Fanuc TP program (LS listing): op5_med_master_air_c.ls

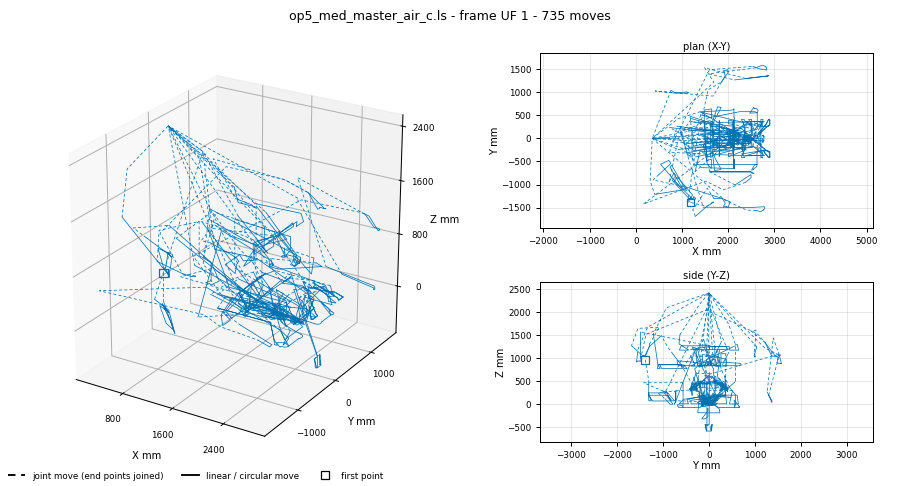
[picture p0: tool path of op5_med_master_air_c.ls in frame UF 1, 735 of 735 moves have a stored position in this frame; points joined in program order, loops and branches not executed]
/PROG  OP5_MED_MASTER_AIR_C
/ATTR
OWNER		= MNEDITOR;
COMMENT		= "Medium Main Air";
PROG_SIZE	= 94128;
CREATE		= DATE 25-08-22  TIME 11:43:26;
MODIFIED	= DATE 26-02-10  TIME 12:20:08;
FILE_NAME	= OP5_MED_;
VERSION		= 0;
LINE_COUNT	= 2444;
MEMORY_SIZE	= 94772;
PROTECT		= READ_WRITE;
TCD:  STACK_SIZE	= 0,
      TASK_PRIORITY	= 50,
      TIME_SLICE	= 0,
      BUSY_LAMP_OFF	= 0,
      ABORT_REQUEST	= 0,
      PAUSE_REQUEST	= 0;
DEFAULT_GROUP	= 1,1,*,*,*;
CONTROL_CODE	= 00000000 00000000;
/APPL
  ARC Welding Equipment : 1,*,*,*,*;

MPAS ;
MPAS_NUM_PASSES        : 0;
MPAS_LAST_PASS         : 0;
MPAS_CURRENT_PASS      : 0;
MPAS_STATUS_PASS       : 0;
/MN
   1:  !********** WAR HAMMER ********** ;
   2:  !*------- FRAME MEIDIUM --------* ;
   3:  !*------- FR500 CELL: C --------* ;
   4:  !******************************** ;
   5:   ;
   6:  CALL HOME    ;
   7:  UFRAME_NUM=1 ;
   8:   ;
   9:  !********POSITIONER MOVE******** ;
  10:J P[1] 85% CNT70    ;
  11:   ;
  12:J P[2] 50% CNT50    ;
  13:   ;
  14:L P[3] 1000mm/sec CNT90    ;
  15:   ;
  16:   ;
  17:  CALL ARC_DISABLE_FRONT_BMPR_MED(0) ;
  18:   ;
  19:  !FR50M1000 ;
  20:  IF R[15]=1001,CALL TECH_HOLD ;
  21:   ;
  22:L P[4] 1000mm/sec FINE
    :  Arc Start[6]    ;
  23:  Weave Sine[6] ;
  24:  Track TAST[6] ;
  25:L P[688] WELD_SPEED CNT100    ;
  26:L P[5] WELD_SPEED FINE
    :  Arc End[6]    ;
  27:  Weave End ;
  28:  Track End ;
  29:   ;
  30:   ;
  31:L P[6] 1000mm/sec CNT100    ;
  32:   ;
  33:L P[7] 1000mm/sec CNT100    ;
  34:   ;
  35:   ;
  36:  !FR50M1001 ;
  37:  IF R[15]=1002,CALL TECH_HOLD ;
  38:   ;
  39:   ;
  40:   ;
  41:L P[8] 1000mm/sec FINE
    :  Arc Start[6]    ;
  42:  Weave Sine[6] ;
  43:  Track TAST[6] ;
  44:L P[9] WELD_SPEED CNT100    ;
  45:L P[12] WELD_SPEED FINE
    :  Arc End[6]    ;
  46:  Weave End ;
  47:  Track End ;
  48:   ;
  49:   ;
  50:L P[10] 1000mm/sec CNT100    ;
  51:   ;
  52:L P[11] 1000mm/sec CNT100    ;
  53:   ;
  54:   ;
  55:  !FR50M1002 ;
  56:  IF R[15]=1003,CALL TECH_HOLD ;
  57:   ;
  58:   ;
  59:   ;
  60:L P[13] 1000mm/sec FINE
    :  Arc Start[6]    ;
  61:  Weave Sine[6] ;
  62:  Track TAST[6] ;
  63:L P[19] WELD_SPEED FINE
    :  Arc End[6]    ;
  64:  Weave End ;
  65:  Track End ;
  66:   ;
  67:   ;
  68:  CALL ARC_DISABLE_FRONT_BMPR_MED(1) ;
  69:   ;
  70:   ;
  71:L P[14] 1000mm/sec CNT80    ;
  72:   ;
  73:  !HOME ;
  74:J P[643] 80% CNT75    ;
  75:   ;
  76:  !********POSITIONER MOVE******** ;
  77:J P[15] 90% CNT40    ;
  78:   ;
  79:J P[16] 70% CNT40    ;
  80:   ;
  81:J P[17] 50% CNT50    ;
  82:   ;
  83:L P[18] 1000mm/sec CNT30    ;
  84:   ;
  85:   ;
  86:  !FR50M1003 ;
  87:  IF R[15]=1004,CALL TECH_HOLD ;
  88:   ;
  89:   ;
  90:   ;
  91:L P[20] 1000mm/sec FINE
    :  Arc Start[6]    ;
  92:  Weave Sine[6] ;
  93:  Track TAST[6] ;
  94:L P[23] WELD_SPEED CNT100    ;
  95:L P[24] WELD_SPEED FINE
    :  Arc End[6]    ;
  96:  Weave End ;
  97:  Track End ;
  98:   ;
  99:   ;
 100:L P[21] 1000mm/sec CNT25    ;
 101:   ;
 102:J P[22] 50% CNT25    ;
 103:   ;
 104:   ;
 105:  !FR50M1010 ;
 106:  IF R[15]=1011,CALL TECH_HOLD ;
 107:   ;
 108:   ;
 109:   ;
 110:L P[27] 1000mm/sec FINE
    :  Arc Start[6]    ;
 111:  Weave Sine[6] ;
 112:  Track TAST[6] ;
 113:L P[28] WELD_SPEED FINE
    :  Arc End[6]    ;
 114:  Weave End ;
 115:  Track End ;
 116:   ;
 117:   ;
 118:L P[25] 1000mm/sec CNT80    ;
 119:   ;
 120:L P[26] 1000mm/sec CNT90    ;
 121:   ;
 122:   ;
 123:  !FR50M1020 ;
 124:  IF R[15]=1021,CALL TECH_HOLD ;
 125:   ;
 126:   ;
 127:   ;
 128:L P[33] 1000mm/sec FINE
    :  Arc Start[6]    ;
 129:  Weave Sine[6] ;
 130:  Track TAST[6] ;
 131:L P[34] WELD_SPEED FINE
    :  Arc End[6]    ;
 132:  Weave End ;
 133:  Track End ;
 134:   ;
 135:   ;
 136:L P[29] 1000mm/sec CNT100    ;
 137:   ;
 138:J P[30] 50% CNT45    ;
 139:   ;
 140:L P[31] 1000mm/sec CNT100    ;
 141:   ;
 142:L P[32] 1000mm/sec CNT30    ;
 143:   ;
 144:   ;
 145:  !FR50M1030 ;
 146:  IF R[15]=1031,CALL TECH_HOLD ;
 147:   ;
 148:   ;
 149:   ;
 150:L P[37] 1000mm/sec FINE
    :  Arc Start[6]    ;
 151:L P[38] WELD_SPEED FINE
    :  Arc End[6]    ;
 152:   ;
 153:   ;
 154:L P[35] 1000mm/sec CNT30    ;
 155:   ;
 156:J P[36] 60% CNT25    ;
 157:   ;
 158:   ;
 159:  !FR50M1040 ;
 160:  IF R[15]=1041,CALL TECH_HOLD ;
 161:   ;
 162:L P[41] 1000mm/sec FINE
    :  Arc Start[6]    ;
 163:L P[42] WELD_SPEED FINE
    :  Arc End[6]    ;
 164:  //L P[47] 1000mm/sec FINE
    :  Arc Start[6]    ;
 165:  //L P[48] WELD_SPEED FINE
    :  Arc End[6]    ;
 166:   ;
 167:   ;
 168:L P[39] 1000mm/sec CNT25    ;
 169:   ;
 170:J P[40] 40% CNT25    ;
 171:   ;
 172:   ;
 173:  !FR50M1050 ;
 174:  IF R[15]=1051,CALL TECH_HOLD ;
 175:   ;
 176:L P[47] 1000mm/sec FINE
    :  Arc Start[6]    ;
 177:L P[687] WELD_SPEED FINE
    :  Arc End[6]    ;
 178:   ;
 179:   ;
 180:  !FR50M1050 ;
 181:  IF R[15]=1051,CALL TECH_HOLD ;
 182:   ;
 183:   ;
 184:L P[43] 500mm/sec CNT75    ;
 185:   ;
 186:L P[44] 1400mm/sec CNT75    ;
 187:   ;
 188:J P[45] 50% CNT25    ;
 189:   ;
 190:L P[46] 1000mm/sec CNT80    ;
 191:   ;
 192:   ;
 193:  !FR50M1060 ;
 194:  IF R[15]=1061,CALL TECH_HOLD ;
 195:   ;
 196:  !50MM ;
 197:   ;
 198:   ;
 199:L P[51] 1000mm/sec FINE
    :  Arc Start[6]    ;
 200:  Weave Sine[6] ;
 201:  Track TAST[6] ;
 202:L P[52] WELD_SPEED FINE
    :  Arc End[6]    ;
 203:  Weave End ;
 204:  Track End ;
 205:   ;
 206:   ;
 207:L P[49] 1000mm/sec CNT90    ;
 208:   ;
 209:L P[50] 1000mm/sec CNT90 Wjnt    ;
 210:   ;
 211:   ;
 212:  !FR50M1070 ;
 213:  IF R[15]=1071,CALL TECH_HOLD ;
 214:   ;
 215:  !50MM ;
 216:   ;
 217:   ;
 218:L P[56] 1000mm/sec FINE
    :  Arc Start[6]    ;
 219:  Weave Sine[6] ;
 220:  Track TAST[6] ;
 221:L P[57] WELD_SPEED FINE
    :  Arc End[6]    ;
 222:  Weave End ;
 223:  Track End ;
 224:   ;
 225:   ;
 226:J P[53] 20% CNT30    ;
 227:   ;
 228:J P[54] 50% CNT25    ;
 229:   ;
 230:L P[55] 1000mm/sec CNT60    ;
 231:   ;
 232:   ;
 233:  !FR50M1080 ;
 234:  IF R[15]=1081,CALL TECH_HOLD ;
 235:   ;
 236:  !10MM PASS ;
 237:   ;
 238:   ;
 239:L P[58] 1000mm/sec FINE
    :  Arc Start[6]    ;
 240:  Weave Sine[6] ;
 241:  Track TAST[6] RPM[1] ;
 242:L P[60] WELD_SPEED CNT100    ;
 243:L P[62] WELD_SPEED CNT100    ;
 244:C P[65]
    :  P[66] WELD_SPEED FINE
    :  Arc End[6]    ;
 245:  Track End ;
 246:  Weave End ;
 247:   ;
 248:   ;
 249:L P[61] 1000mm/sec CNT60    ;
 250:   ;
 251:L P[59] 1000mm/sec CNT100    ;
 252:   ;
 253:J P[63] 50% CNT40    ;
 254:   ;
 255:L P[64] 1000mm/sec CNT50    ;
 256:   ;
 257:  !FR50M1090 ;
 258:  IF R[15]=1091,CALL TECH_HOLD ;
 259:   ;
 260:  !10MM PASS ;
 261:   ;
 262:   ;
 263:L P[67] 1000mm/sec FINE
    :  Arc Start[6]    ;
 264:  Weave Sine[6] ;
 265:  Track TAST[6] RPM[2] ;
 266:L P[69] WELD_SPEED CNT100    ;
 267:L P[72] WELD_SPEED CNT100    ;
 268:C P[75]
    :  P[77] WELD_SPEED FINE
    :  Arc End[6]    ;
 269:  Track End ;
 270:  Weave End ;
 271:   ;
 272:   ;
 273:L P[70] 500mm/sec CNT50    ;
 274:   ;
 275:J P[68] 50% CNT35    ;
 276:   ;
 277:J P[71] 50% CNT25    ;
 278:   ;
 279:   ;
 280:  !FR50M1081 ;
 281:  IF R[15]=1082,CALL TECH_HOLD ;
 282:   ;
 283:   ;
 284:L P[74] 1000mm/sec CNT40    ;
 285:   ;
 286:  MP Offset  PR[3] RPM[1] ;
 287:   ;
 288:L P[58] 1000mm/sec FINE
    :  Arc Start[6]    ;
 289:  Weave Sine[6] ;
 290:L P[60] WELD_SPEED CNT100    ;
 291:L P[62] WELD_SPEED CNT100    ;
 292:C P[65]
    :  P[66] WELD_SPEED FINE
    :  Arc End[6]    ;
 293:  Weave End ;
 294:   ;
 295:  MP Offset End ;
 296:   ;
 297:L P[80] 1000mm/sec CNT40    ;
 298:   ;
 299:L P[685] 500mm/sec CNT100    ;
 300:   ;
 301:   ;
 302:  !FR50M1082 ;
 303:  IF R[15]=1083,CALL TECH_HOLD ;
 304:   ;
 305:   ;
 306:J P[81] 50% CNT30    ;
 307:   ;
 308:L P[82] 1000mm/sec CNT30    ;
 309:   ;
 310:  MP Offset  PR[4] RPM[1] ;
 311:   ;
 312:L P[58] 1000mm/sec FINE
    :  Arc Start[6]    ;
 313:  Weave Sine[6] ;
 314:L P[60] WELD_SPEED CNT100    ;
 315:L P[62] WELD_SPEED CNT100    ;
 316:C P[65]
    :  P[66] WELD_SPEED FINE
    :  Arc End[6]    ;
 317:  Weave End ;
 318:   ;
 319:  MP Offset End ;
 320:   ;
 321:L P[83] 1000mm/sec CNT25    ;
 322:   ;
 323:L P[84] 500mm/sec CNT100    ;
 324:   ;
 325:   ;
 326:  !FR50M1091 ;
 327:  IF R[15]=1092,CALL TECH_HOLD ;
 328:   ;
 329:   ;
 330:J P[85] 50% CNT25    ;
 331:   ;
 332:L P[86] 1000mm/sec CNT50    ;
 333:   ;
 334:  MP Offset  PR[1] RPM[2] ;
 335:   ;
 336:L P[67] 1000mm/sec FINE
    :  Arc Start[6]    ;
 337:  Weave Sine[6] ;
 338:L P[69] WELD_SPEED CNT100    ;
 339:L P[72] WELD_SPEED CNT100    ;
 340:C P[75]
    :  P[77] WELD_SPEED FINE
    :  Arc End[6]    ;
 341:  Weave End ;
 342:   ;
 343:  MP Offset End ;
 344:   ;
 345:L P[87] 500mm/sec CNT30    ;
 346:   ;
 347:J P[88] 50% CNT25    ;
 348:   ;
 349:   ;
 350:  !FR50M1092 ;
 351:  IF R[15]=1093,CALL TECH_HOLD ;
 352:   ;
 353:   ;
 354:L P[89] 1000mm/sec CNT50    ;
 355:   ;
 356:  MP Offset  PR[2] RPM[2] ;
 357:   ;
 358:L P[67] 1000mm/sec FINE
    :  Arc Start[6]    ;
 359:  Weave Sine[6] ;
 360:L P[69] WELD_SPEED CNT100    ;
 361:L P[72] WELD_SPEED CNT100    ;
 362:C P[75]
    :  P[77] WELD_SPEED FINE
    :  Arc End[6]    ;
 363:  Weave End ;
 364:   ;
 365:  MP Offset End ;
 366:   ;
 367:L P[90] 500mm/sec CNT50    ;
 368:   ;
 369:J P[102] 50% CNT25    ;
 370:   ;
 371:L P[103] 1000mm/sec CNT80    ;
 372:   ;
 373:   ;
 374:  !FR50M1100 ;
 375:  IF R[15]=1101,CALL TECH_HOLD ;
 376:   ;
 377:   ;
 378:   ;
 379:L P[124] 1000mm/sec FINE
    :  Arc Start[8]    ;
 380:  Weave Sine[8] ;
 381:L P[128] WELD_SPEED CNT100    ;
 382:C P[129]
    :  P[132] WELD_SPEED FINE
    :  Arc End[8]    ;
 383:  Weave End ;
 384:   ;
 385:   ;
 386:L P[108] 1000mm/sec CNT40    ;
 387:   ;
 388:L P[109] 1000mm/sec CNT30    ;
 389:   ;
 390:J P[110] 50% CNT30    ;
 391:   ;
 392:L P[111] 1000mm/sec CNT80    ;
 393:   ;
 394:   ;
 395:  !FR50M1110 ;
 396:  IF R[15]=1111,CALL TECH_HOLD ;
 397:   ;
 398:   ;
 399:   ;
 400:L P[133] 1000mm/sec FINE
    :  Arc Start[8]    ;
 401:  Weave Sine[8] ;
 402:L P[138] WELD_SPEED CNT100    ;
 403:C P[139]
    :  P[142] WELD_SPEED FINE
    :  Arc End[8]    ;
 404:  Weave End ;
 405:   ;
 406:   ;
 407:L P[116] 1000mm/sec CNT40    ;
 408:   ;
 409:J P[117] 50% CNT40    ;
 410:   ;
 411:L P[118] 1000mm/sec CNT80    ;
 412:   ;
 413:   ;
 414:  !FR50M1120 ;
 415:  !75mm ;
 416:  IF R[15]=1121,CALL TECH_HOLD ;
 417:   ;
 418:   ;
 419:   ;
 420:L P[143] 1000mm/sec FINE
    :  Arc Start[6]    ;
 421:  Weave Sine[6] ;
 422:  Track TAST[6] ;
 423:L P[145] WELD_SPEED FINE
    :  Arc End[6]    ;
 424:  Weave End ;
 425:  Track End ;
 426:   ;
 427:   ;
 428:L P[121] 1000mm/sec CNT90    ;
 429:   ;
 430:L P[122] 1000mm/sec CNT80    ;
 431:   ;
 432:   ;
 433:  !FR50M1130 ;
 434:  IF R[15]=1131,CALL TECH_HOLD ;
 435:   ;
 436:  !75mm ;
 437:   ;
 438:   ;
 439:L P[146] 1000mm/sec FINE
    :  Arc Start[6]    ;
 440:  Weave Sine[6] ;
 441:  Track TAST[6] ;
 442:L P[149] WELD_SPEED FINE
    :  Arc End[6]    ;
 443:  Weave End ;
 444:  Track End ;
 445:   ;
 446:   ;
 447:L P[125] 1000mm/sec CNT100    ;
 448:   ;
 449:L P[126] 1000mm/sec CNT100    ;
 450:   ;
 451:  !********POSITIONER MOVE******** ;
 452:J P[127] 75% CNT30    ;
 453:   ;
 454:   ;
 455:   ;
 456:  !FR50M1140 ;
 457:  IF R[15]=1141,CALL TECH_HOLD ;
 458:   ;
 459:L P[150] 1000mm/sec FINE
    :  Arc Start[6]    ;
 460:  Weave Sine[6] ;
 461:  Track TAST[6] ;
 462:L P[156] WELD_SPEED FINE
    :  Arc End[6]    ;
 463:  Weave End ;
 464:  Track End ;
 465:   ;
 466:   ;
 467:L P[130] 1000mm/sec CNT90    ;
 468:   ;
 469:L P[131] 1000mm/sec CNT60    ;
 470:   ;
 471:   ;
 472:  !FR50M1150 ;
 473:  IF R[15]=1151,CALL TECH_HOLD ;
 474:   ;
 475:   ;
 476:   ;
 477:L P[157] 1000mm/sec FINE
    :  Arc Start[6]    ;
 478:  Weave Sine[6] ;
 479:  Track TAST[6] ;
 480:L P[158] WELD_SPEED FINE
    :  Arc End[6]    ;
 481:  Weave End ;
 482:  Track End ;
 483:   ;
 484:   ;
 485:L P[134] 1000mm/sec CNT90    ;
 486:   ;
 487:  !HOME ;
 488:J P[756] 100% CNT90    ;
 489:   ;
 490:  !********POSITIONER MOVE******** ;
 491:J P[135] 85% CNT50    ;
 492:   ;
 493:J P[136] 50% CNT40    ;
 494:   ;
 495:L P[137] 1000mm/sec CNT30    ;
 496:   ;
 497:   ;
 498:  !FR50M1160 ;
 499:  IF R[15]=1161,CALL TECH_HOLD ;
 500:   ;
 501:   ;
 502:   ;
 503:L P[162] 350mm/sec FINE
    :  Arc Start[6]    ;
 504:  Weave Sine[6] ;
 505:  Track TAST[6] ;
 506:L P[163] WELD_SPEED CNT100    ;
 507:L P[164] WELD_SPEED FINE
    :  Arc End[6]    ;
 508:  Weave End ;
 509:  Track End ;
 510:   ;
 511:   ;
 512:L P[140] 800mm/sec CNT30    ;
 513:   ;
 514:L P[141] 1000mm/sec CNT30    ;
 515:   ;
 516:   ;
 517:  !FR50M1170 ;
 518:  IF R[15]=1171,CALL TECH_HOLD ;
 519:   ;
 520:   ;
 521:   ;
 522:L P[78] 400mm/sec FINE
    :  Arc Start[6]    ;
 523:  Weave Sine[6] ;
 524:  Track TAST[6] ;
 525:L P[79] WELD_SPEED FINE
    :  Arc End[6]    ;
 526:  Weave End ;
 527:  Track End ;
 528:   ;
 529:   ;
 530:L P[144] 700mm/sec CNT50    ;
 531:   ;
 532:L P[73] 1000mm/sec CNT50    ;
 533:   ;
 534:   ;
 535:  !FR50M1180 ;
 536:  IF R[15]=1181,CALL TECH_HOLD ;
 537:   ;
 538:   ;
 539:   ;
 540:L P[172] 500mm/sec FINE
    :  Arc Start[6]    ;
 541:  Weave Sine[6] ;
 542:  Track TAST[6] ;
 543:L P[173] WELD_SPEED FINE
    :  Arc End[6]    ;
 544:  Weave End ;
 545:  Track End ;
 546:   ;
 547:   ;
 548:L P[147] 600mm/sec CNT60    ;
 549:   ;
 550:L P[148] 1200mm/sec CNT35    ;
 551:   ;
 552:   ;
 553:  !FR50M1190 ;
 554:  IF R[15]=1191,CALL TECH_HOLD ;
 555:   ;
 556:   ;
 557:   ;
 558:L P[176] 100mm/sec FINE
    :  Arc Start[6]    ;
 559:  Weave Sine[6] ;
 560:  Track TAST[6] ;
 561:L P[177] WELD_SPEED CNT100    ;
 562:L P[180] WELD_SPEED FINE
    :  Arc End[6]    ;
 563:  Weave End ;
 564:  Track End ;
 565:   ;
 566:   ;
 567:L P[151] 500mm/sec CNT50    ;
 568:   ;
 569:L P[152] 1000mm/sec CNT90    ;
 570:   ;
 571:J P[757] 100% CNT40    ;
 572:   ;
 573:  !********POSITIONER MOVE******** ;
 574:J P[153] 85% CNT25    ;
 575:   ;
 576:  CALL HOME    ;
 577:  CALL T_CLEAN    ;
 578:   ;
 579:J P[154] 50% CNT45    ;
 580:   ;
 581:L P[155] 1000mm/sec CNT35    ;
 582:   ;
 583:L P[76] 800mm/sec CNT25    ;
 584:   ;
 585:   ;
 586:  !FR50M1200 ;
 587:  IF R[15]=1201,CALL TECH_HOLD ;
 588:   ;
 589:   ;
 590:L P[181] 1000mm/sec FINE
    :  Arc Start[6]    ;
 591:  Weave Sine[6] ;
 592:  Track TAST[6] ;
 593:L P[184] WELD_SPEED CNT100    ;
 594:L P[185] WELD_SPEED CNT100    ;
 595:L P[190] WELD_SPEED FINE
    :  Arc End[6]    ;
 596:  Weave End ;
 597:  Track End ;
 598:   ;
 599:   ;
 600:L P[159] 1000mm/sec CNT25    ;
 601:   ;
 602:J P[160] 50% CNT35    ;
 603:   ;
 604:L P[161] 1000mm/sec CNT45    ;
 605:   ;
 606:   ;
 607:  !FR50M1210 ;
 608:  IF R[15]=1211,CALL TECH_HOLD ;
 609:   ;
 610:   ;
 611:   ;
 612:L P[191] 1000mm/sec FINE
    :  Arc Start[6]    ;
 613:  Weave Sine[6] ;
 614:  Track TAST[6] ;
 615:L P[194] WELD_SPEED CNT100    ;
 616:L P[195] WELD_SPEED CNT100    ;
 617:L P[197] WELD_SPEED FINE
    :  Arc End[6]    ;
 618:  Weave End ;
 619:  Track End ;
 620:   ;
 621:   ;
 622:L P[165] 500mm/sec CNT50    ;
 623:   ;
 624:J P[166] 50% CNT35    ;
 625:   ;
 626:L P[167] 1000mm/sec CNT50    ;
 627:   ;
 628:   ;
 629:  !FR50M1220 ;
 630:  IF R[15]=1221,CALL TECH_HOLD ;
 631:   ;
 632:  //UALM[20] ;
 633:   ;
 634:L P[198] 1000mm/sec FINE
    :  Arc Start[6]    ;
 635:  Weave Sine[6] ;
 636:  Track TAST[6] ;
 637:L P[205] WELD_SPEED CNT100    ;
 638:L P[206] WELD_SPEED FINE
    :  Arc End[6]    ;
 639:  Weave End ;
 640:  Track End ;
 641:   ;
 642:   ;
 643:L P[92] 1000mm/sec CNT100    ;
 644:   ;
 645:L P[170] 1400mm/sec CNT80    ;
 646:   ;
 647:L P[171] 1000mm/sec CNT50    ;
 648:   ;
 649:   ;
 650:  !FR50M1230 ;
 651:  IF R[15]=1231,CALL TECH_HOLD ;
 652:   ;
 653:   ;
 654:   ;
 655:L P[209] 1000mm/sec FINE
    :  Arc Start[6]    ;
 656:  Weave Sine[6] ;
 657:  Track TAST[6] ;
 658:L P[210] WELD_SPEED CNT100    ;
 659:L P[215] WELD_SPEED FINE
    :  Arc End[6]    ;
 660:  Weave End ;
 661:  Track End ;
 662:   ;
 663:   ;
 664:L P[174] 1000mm/sec CNT80    ;
 665:   ;
 666:L P[175] 1000mm/sec CNT90    ;
 667:   ;
 668:   ;
 669:  !FR50M1240 ;
 670:  IF R[15]=1241,CALL TECH_HOLD ;
 671:   ;
 672:   ;
 673:   ;
 674:L P[216] 1000mm/sec FINE
    :  Arc Start[6]    ;
 675:  Weave Sine[6] ;
 676:  Track TAST[6] ;
 677:L P[217] WELD_SPEED FINE
    :  Arc End[6]    ;
 678:  Weave End ;
 679:  Track End ;
 680:   ;
 681:   ;
 682:L P[178] 1000mm/sec CNT80    ;
 683:   ;
 684:L P[179] 1000mm/sec CNT90    ;
 685:   ;
 686:   ;
 687:  !FR50M1250 ;
 688:  IF R[15]=1251,CALL TECH_HOLD ;
 689:   ;
 690:   ;
 691:   ;
 692:L P[218] 1000mm/sec FINE
    :  Arc Start[6]    ;
 693:  Weave Sine[6] ;
 694:  Track TAST[6] ;
 695:L P[221] WELD_SPEED FINE
    :  Arc End[6]    ;
 696:  Weave End ;
 697:  Track End ;
 698:   ;
 699:   ;
 700:L P[182] 1000mm/sec CNT90    ;
 701:   ;
 702:L P[183] 1300mm/sec CNT80    ;
 703:   ;
 704:   ;
 705:  !FR50M1260 ;
 706:  IF R[15]=1261,CALL TECH_HOLD ;
 707:   ;
 708:   ;
 709:   ;
 710:L P[222] 1000mm/sec FINE
    :  Arc Start[6]    ;
 711:  Weave Sine[6] ;
 712:  Track TAST[6] ;
 713:L P[224] WELD_SPEED CNT100    ;
 714:L P[225] WELD_SPEED FINE
    :  Arc End[6]    ;
 715:  Weave End ;
 716:  Track End ;
 717:   ;
 718:   ;
 719:L P[186] 1000mm/sec CNT80    ;
 720:   ;
 721:J P[187] 50% CNT30    ;
 722:   ;
 723:  !********POSITIONER MOVE******** ;
 724:J P[188] 80% CNT30    ;
 725:   ;
 726:L P[189] 1000mm/sec CNT35    ;
 727:   ;
 728:   ;
 729:  !FR50M1270 ;
 730:  IF R[15]=1271,CALL TECH_HOLD ;
 731:   ;
 732:   ;
 733:L P[228] 1000mm/sec FINE
    :  Arc Start[8]    ;
 734:  Weave Sine[8] ;
 735:L P[229] WELD_SPEED FINE
    :  Arc End[8]    ;
 736:  Weave End ;
 737:   ;
 738:   ;
 739:L P[192] 1000mm/sec CNT40    ;
 740:   ;
 741:J P[759] 100% CNT30    ;
 742:   ;
 743:  !********POSITIONER MOVE******** ;
 744:J P[193] 85% CNT30    ;
 745:   ;
 746:   ;
 747:  !FR50M1280 ;
 748:  IF R[15]=1281,CALL TECH_HOLD ;
 749:   ;
 750:   ;
 751:   ;
 752:L P[232] 1000mm/sec FINE
    :  Arc Start[6]    ;
 753:  Weave Sine[6] ;
 754:L P[233] WELD_SPEED FINE
    :  Arc End[6]    ;
 755:  Weave End ;
 756:   ;
 757:   ;
 758:   ;
 759:  !FR50M1290 ;
 760:  IF R[15]=1291,CALL TECH_HOLD ;
 761:   ;
 762:   ;
 763:L P[196] 1000mm/sec CNT100    ;
 764:   ;
 765:   ;
 766:L P[236] 1000mm/sec FINE
    :  Arc Start[6]    ;
 767:  Weave Sine[6] ;
 768:L P[238] WELD_SPEED FINE
    :  Arc End[6]    ;
 769:  Weave End ;
 770:   ;
 771:   ;
 772:L P[199] 1000mm/sec CNT75    ;
 773:   ;
 774:J P[94] 50% CNT100    ;
 775:   ;
 776:J P[200] 50% CNT100    ;
 777:   ;
 778:  !HOME ;
 779:J P[760] 60% CNT30    ;
 780:   ;
 781:  !********POSITIONER MOVE******** ;
 782:J P[201] 85% CNT25    ;
 783:   ;
 784:L P[203] 1200mm/sec CNT25    ;
 785:   ;
 786:L P[204] 1000mm/sec CNT25    ;
 787:   ;
 788:   ;
 789:  !FR50M1300 ;
 790:  IF R[15]=1301,CALL TECH_HOLD ;
 791:   ;
 792:   ;
 793:   ;
 794:L P[239] 1000mm/sec FINE
    :  Arc Start[6]    ;
 795:  Weave Sine[6] ;
 796:  Track TAST[6] ;
 797:L P[240] WELD_SPEED CNT100    ;
 798:L P[241] WELD_SPEED FINE
    :  Arc End[6]    ;
 799:  Weave End ;
 800:  Track End ;
 801:   ;
 802:   ;
 803:L P[207] 1000mm/sec CNT25    ;
 804:   ;
 805:J P[208] 50% CNT25    ;
 806:   ;
 807:   ;
 808:  !FR50M1310 ;
 809:  IF R[15]=1311,CALL TECH_HOLD ;
 810:   ;
 811:   ;
 812:L P[246] 1000mm/sec FINE
    :  Arc Start[6]    ;
 813:  Weave Sine[6] ;
 814:  Track TAST[6] ;
 815:L P[247] WELD_SPEED CNT100    ;
 816:L P[249] WELD_SPEED CNT100    ;
 817:L P[250] WELD_SPEED FINE
    :  Arc End[6]    ;
 818:  Weave End ;
 819:  Track End ;
 820:   ;
 821:   ;
 822:L P[211] 1000mm/sec CNT25    ;
 823:   ;
 824:L P[212] 1000mm/sec CNT25    ;
 825:   ;
 826:L P[213] 1000mm/sec CNT25    ;
 827:   ;
 828:  !********POSITIONER MOVE******** ;
 829:J P[214] 75% CNT10    ;
 830:   ;
 831:   ;
 832:  !FR50M1320 ;
 833:  IF R[15]=1321,CALL TECH_HOLD ;
 834:   ;
 835:   ;
 836:   ;
 837:L P[253] 1000mm/sec FINE
    :  Arc Start[6]    ;
 838:  Weave Sine[6] ;
 839:L P[254] WELD_SPEED CNT100    ;
 840:L P[255] WELD_SPEED CNT100    ;
 841:L P[258] WELD_SPEED FINE
    :  Arc End[6]    ;
 842:  Weave End ;
 843:   ;
 844:   ;
 845:L P[219] 1000mm/sec CNT40    ;
 846:   ;
 847:L P[220] 1000mm/sec CNT40    ;
 848:   ;
 849:   ;
 850:  !FR50M1330 ;
 851:  IF R[15]=1331,CALL TECH_HOLD ;
 852:   ;
 853:   ;
 854:   ;
 855:L P[259] 1000mm/sec FINE
    :  Arc Start[6]    ;
 856:  Weave Sine[6] ;
 857:  Track TAST[6] ;
 858:L P[264] WELD_SPEED FINE
    :  Arc End[6]    ;
 859:  Weave End ;
 860:  Track End ;
 861:   ;
 862:   ;
 863:L P[223] 1000mm/sec CNT30    ;
 864:   ;
 865:   ;
 866:  !FR50M1340 ;
 867:  IF R[15]=1341,CALL TECH_HOLD ;
 868:   ;
 869:   ;
 870:   ;
 871:L P[265] 1000mm/sec FINE
    :  Arc Start[6]    ;
 872:  Weave Sine[6] ;
 873:  Track TAST[6] ;
 874:L P[269] WELD_SPEED CNT100    ;
 875:L P[270] WELD_SPEED FINE
    :  Arc End[6]    ;
 876:  Weave End ;
 877:  Track End ;
 878:   ;
 879:   ;
 880:L P[226] 1000mm/sec CNT30    ;
 881:   ;
 882:L P[227] 1000mm/sec CNT25    ;
 883:   ;
 884:L P[99] 1000mm/sec CNT40    ;
 885:   ;
 886:   ;
 887:  !FR50M1350 ;
 888:  IF R[15]=1351,CALL TECH_HOLD ;
 889:   ;
 890:   ;
 891:   ;
 892:L P[273] 1000mm/sec FINE
    :  Arc Start[6]    ;
 893:  Weave Sine[6] ;
 894:  Track TAST[6] ;
 895:L P[274] WELD_SPEED CNT100    ;
 896:L P[279] WELD_SPEED CNT100    ;
 897:L P[280] WELD_SPEED FINE
    :  Arc End[6]    ;
 898:  Weave End ;
 899:  Track End ;
 900:   ;
 901:   ;
 902:L P[230] 1000mm/sec CNT40    ;
 903:   ;
 904:J P[231] 50% CNT25    ;
 905:   ;
 906:   ;
 907:  !FR50M1360 ;
 908:  IF R[15]=1361,CALL TECH_HOLD ;
 909:   ;
 910:   ;
 911:   ;
 912:L P[281] 1000mm/sec FINE
    :  Arc Start[6]    ;
 913:  Weave Sine[6] ;
 914:  Track TAST[6] ;
 915:L P[282] WELD_SPEED CNT100    ;
 916:L P[283] WELD_SPEED FINE
    :  Arc End[6]    ;
 917:  Weave End ;
 918:  Track End ;
 919:   ;
 920:   ;
 921:L P[234] 1000mm/sec CNT25    ;
 922:   ;
 923:J P[235] 50% CNT25    ;
 924:   ;
 925:   ;
 926:  !FR50M1370 ;
 927:  IF R[15]=1371,CALL TECH_HOLD ;
 928:   ;
 929:   ;
 930:   ;
 931:L P[284] 1000mm/sec FINE
    :  Arc Start[6]    ;
 932:  Weave Sine[6] ;
 933:L P[285] WELD_SPEED CNT100    ;
 934:L P[286] WELD_SPEED FINE
    :  Arc End[6]    ;
 935:   ;
 936:   ;
 937:L P[237] 1000mm/sec CNT25    ;
 938:   ;
 939:   ;
 940:  !FR50M1380 ;
 941:  IF R[15]=1381,CALL TECH_HOLD ;
 942:   ;
 943:   ;
 944:   ;
 945:L P[287] 1000mm/sec FINE
    :  Arc Start[6]    ;
 946:  Weave Sine[6] ;
 947:L P[288] WELD_SPEED CNT100    ;
 948:  Weave End ;
 949:L P[289] WELD_SPEED FINE
    :  Arc End[6]    ;
 950:   ;
 951:   ;
 952:L P[242] 1000mm/sec CNT100    ;
 953:   ;
 954:L P[243] 1000mm/sec CNT100    ;
 955:   ;
 956:J P[244] 50% CNT40    ;
 957:   ;
 958:L P[245] 1000mm/sec CNT25    ;
 959:   ;
 960:   ;
 961:  !FR50M1390 ;
 962:  IF R[15]=1391,CALL TECH_HOLD ;
 963:   ;
 964:   ;
 965:   ;
 966:L P[293] 1000mm/sec FINE
    :  Arc Start[6]    ;
 967:  Weave Sine[6] ;
 968:  Track TAST[6] ;
 969:L P[294] WELD_SPEED FINE
    :  Arc End[6]    ;
 970:  Weave End ;
 971:  Track End ;
 972:   ;
 973:   ;
 974:L P[248] 1000mm/sec CNT25    ;
 975:   ;
 976:   ;
 977:  !FR50M1400 ;
 978:  IF R[15]=1401,CALL TECH_HOLD ;
 979:   ;
 980:   ;
 981:   ;
 982:L P[298] 1000mm/sec FINE
    :  Arc Start[6]    ;
 983:  Weave Sine[6] ;
 984:  Track TAST[6] ;
 985:L P[299] WELD_SPEED CNT100    ;
 986:L P[301] WELD_SPEED FINE
    :  Arc End[6]    ;
 987:  Weave End ;
 988:  Track End ;
 989:   ;
 990:   ;
 991:L P[251] 1000mm/sec CNT100    ;
 992:   ;
 993:L P[252] 1000mm/sec CNT25    ;
 994:   ;
 995:   ;
 996:  !FR50M1410 ;
 997:  IF R[15]=1411,CALL TECH_HOLD ;
 998:   ;
 999:   ;
1000:   ;
1001:L P[302] 1000mm/sec FINE
    :  Arc Start[6]    ;
1002:  Weave Sine[6] ;
1003:  Track TAST[6] ;
1004:L P[309] WELD_SPEED CNT100    ;
1005:L P[310] WELD_SPEED FINE
    :  Arc End[6]    ;
1006:  Weave End ;
1007:  Track End ;
1008:   ;
1009:   ;
1010:L P[256] 1000mm/sec CNT25    ;
1011:   ;
1012:  !********POSITIONER MOVE******** ;
1013:J P[257] 75% FINE    ;
1014:   ;
1015:   ;
1016:  !FR50M1420 ;
1017:  IF R[15]=1421,CALL TECH_HOLD ;
1018:   ;
1019:   ;
1020:   ;
1021:L P[311] 1000mm/sec FINE
    :  Arc Start[6]    ;
1022:  Weave Sine[6] ;
1023:  Track TAST[6] ;
1024:L P[312] WELD_SPEED FINE
    :  Arc End[6]    ;
1025:  Weave End ;
1026:  Track End ;
1027:   ;
1028:   ;
1029:L P[260] 1000mm/sec CNT25    ;
1030:   ;
1031:L P[261] 500mm/sec FINE    ;
1032:   ;
1033:  !********POSITIONER MOVE******** ;
1034:J P[262] 50% CNT25    ;
1035:   ;
1036:L P[263] 1000mm/sec CNT25    ;
1037:   ;
1038:   ;
1039:  !FR50M1430 ;
1040:  IF R[15]=1431,CALL TECH_HOLD ;
1041:   ;
1042:   ;
1043:   ;
1044:L P[313] 1000mm/sec FINE
    :  Arc Start[6]    ;
1045:  Weave Sine[6] ;
1046:L P[314] WELD_SPEED CNT100    ;
1047:L P[315] WELD_SPEED FINE
    :  Arc End[6]    ;
1048:  Weave End ;
1049:   ;
1050:   ;
1051:L P[266] 1000mm/sec CNT25    ;
1052:   ;
1053:L P[690] 1000mm/sec CNT25    ;
1054:   ;
1055:  !********POSITIONER MOVE******** ;
1056:J P[267] 75% CNT25    ;
1057:   ;
1058:L P[268] 1000mm/sec CNT25    ;
1059:   ;
1060:   ;
1061:  !FR50M1440 ;
1062:  IF R[15]=1441,CALL TECH_HOLD ;
1063:   ;
1064:   ;
1065:   ;
1066:L P[316] 1000mm/sec FINE
    :  Arc Start[8]    ;
1067:  Weave Sine[8] ;
1068:L P[322] WELD_SPEED FINE
    :  Arc End[8]    ;
1069:  Weave End ;
1070:   ;
1071:   ;
1072:L P[271] 1000mm/sec CNT25    ;
1073:   ;
1074:L P[272] 500mm/sec CNT25    ;
1075:   ;
1076:  !FR50M1450 ;
1077:  IF R[15]=1451,CALL TECH_HOLD ;
1078:   ;
1079:   ;
1080:L P[323] 1000mm/sec FINE
    :  Arc Start[6]    ;
1081:  Weave Sine[6] ;
1082:  Track TAST[6] ;
1083:L P[324] WELD_SPEED FINE
    :  Arc End[6]    ;
1084:  Weave End ;
1085:  Track End ;
1086:   ;
1087:   ;
1088:L P[275] 1000mm/sec CNT25    ;
1089:   ;
1090:L P[276] 1300mm/sec CNT100    ;
1091:   ;
1092:J P[761] 60% CNT25    ;
1093:   ;
1094:  !********POSITIONER MOVE******** ;
1095:J P[277] 75% CNT25    ;
1096:   ;
1097:L P[278] 1000mm/sec CNT40    ;
1098:   ;
1099:   ;
1100:  !FR50M1460 ;
1101:  IF R[15]=1461,CALL TECH_HOLD ;
1102:   ;
1103:   ;
1104:   ;
1105:L P[325] 1000mm/sec FINE
    :  Arc Start[6]    ;
1106:  Weave Sine[6] ;
1107:  Track TAST[6] ;
1108:L P[326] WELD_SPEED CNT100    ;
1109:C P[327]
    :  P[330] WELD_SPEED CNT100    ;
1110:L P[331] WELD_SPEED CNT100    ;
1111:C P[332]
    :  P[333] WELD_SPEED CNT100    ;
1112:L P[339] WELD_SPEED CNT100    ;
1113:C P[340]
    :  P[341] WELD_SPEED CNT100    ;
1114:L P[342] WELD_SPEED FINE
    :  Arc End[6]    ;
1115:  Weave End ;
1116:  Track End ;
1117:   ;
1118:   ;
1119:L P[290] 1000mm/sec CNT100    ;
1120:   ;
1121:J P[777] 50% CNT50    ;
1122:   ;
1123:J P[291] 50% CNT50    ;
1124:   ;
1125:L P[292] 1000mm/sec CNT25    ;
1126:   ;
1127:   ;
1128:  !FR50M1470 ;
1129:  IF R[15]=1471,CALL TECH_HOLD ;
1130:   ;
1131:   ;
1132:   ;
1133:L P[356] 1000mm/sec FINE
    :  Arc Start[6]    ;
1134:  Weave Sine[6] ;
1135:  Track TAST[6] ;
1136:L P[359] WELD_SPEED FINE
    :  Arc End[6]    ;
1137:  Weave End ;
1138:  Track End ;
1139:   ;
1140:   ;
1141:L P[691] 1000mm/sec CNT25    ;
1142:   ;
1143:L P[295] 1000mm/sec CNT100    ;
1144:   ;
1145:J P[296] 100% CNT25    ;
1146:   ;
1147:L P[297] 1000mm/sec CNT25    ;
1148:   ;
1149:   ;
1150:  !FR50M1480 ;
1151:  IF R[15]=1481,CALL TECH_HOLD ;
1152:   ;
1153:   ;
1154:   ;
1155:L P[360] 1000mm/sec FINE
    :  Arc Start[6]    ;
1156:  Weave Sine[6] ;
1157:  Track TAST[6] ;
1158:L P[368] WELD_SPEED FINE
    :  Arc End[6]    ;
1159:  Weave End ;
1160:  Track End ;
1161:   ;
1162:   ;
1163:L P[300] 1000mm/sec CNT25    ;
1164:   ;
1165:L P[692] 1000mm/sec CNT25    ;
1166:   ;
1167:   ;
1168:  !FR50M1490 ;
1169:  IF R[15]=1491,CALL TECH_HOLD ;
1170:   ;
1171:   ;
1172:   ;
1173:L P[369] 1000mm/sec FINE
    :  Arc Start[6]    ;
1174:  Weave Sine[6] ;
1175:  Track TAST[6] ;
1176:L P[370] WELD_SPEED CNT100    ;
1177:L P[375] WELD_SPEED FINE
    :  Arc End[6]    ;
1178:  Weave End ;
1179:  Track End ;
1180:   ;
1181:   ;
1182:L P[303] 1000mm/sec CNT25    ;
1183:   ;
1184:L P[304] 1000mm/sec CNT100    ;
1185:   ;
1186:J P[305] 50% CNT25    ;
1187:   ;
1188:  !********POSITIONER MOVE******** ;
1189:J P[306] 50% CNT25    ;
1190:   ;
1191:J P[307] 60% CNT25    ;
1192:   ;
1193:  CALL ARC_DISABLE_RH_LS(0) ;
1194:   ;
1195:   ;
1196:  !FR50M1500 ;
1197:  IF R[15]=1501,CALL TECH_HOLD ;
1198:   ;
1199:   ;
1200:L P[308] 1000mm/sec CNT30    ;
1201:   ;
1202:   ;
1203:L P[376] 1000mm/sec FINE
    :  Arc Start[8]    ;
1204:  Weave Sine[8] ;
1205:L P[382] WELD_SPEED CNT100    ;
1206:C P[383]
    :  P[384] WELD_SPEED CNT100    ;
1207:L P[385] WELD_SPEED CNT100    ;
1208:L P[386] WELD_SPEED CNT100    ;
1209:L P[387] WELD_SPEED CNT100    ;
1210:L P[388] WELD_SPEED FINE
    :  Arc End[8]    ;
1211:  Weave End ;
1212:   ;
1213:   ;
1214:  CALL ARC_DISABLE_RH_LS(1) ;
1215:   ;
1216:L P[317] 1000mm/sec CNT40    ;
1217:   ;
1218:J P[318] 45% CNT95    ;
1219:   ;
1220:J P[631] 50% CNT25    ;
1221:   ;
1222:L P[632] 3000mm/sec CNT25    ;
1223:   ;
1224:  !CELL ID: C ... ;
1225:   ;
1226:L P[363] 1000mm/sec CNT100    ;
1227:   ;
1228:L P[93] 800mm/sec FINE
    :  Arc Start[1]    ;
1229:  WAIT    .20(sec) ;
1230:L P[93] WELD_SPEED FINE
    :  Arc End[1]    ;
1231:   ;
1232:L P[96] 800mm/sec FINE
    :  Arc Start[1]    ;
1233:  WAIT    .20(sec) ;
1234:L P[96] WELD_SPEED FINE
    :  Arc End[1]    ;
1235:   ;
1236:L P[98] 800mm/sec FINE
    :  Arc Start[1]    ;
1237:  WAIT    .20(sec) ;
1238:L P[98] WELD_SPEED FINE
    :  Arc End[1]    ;
1239:   ;
1240:L P[634] 1000mm/sec CNT100    ;
1241:   ;
1242:L P[635] 1000mm/sec CNT25    ;
1243:   ;
1244:J P[636] 50% CNT100    ;
1245:   ;
1246:J P[425] 50% CNT70    ;
1247:   ;
1248:  !HOME ;
1249:J P[762] 100% CNT40    ;
1250:   ;
1251:  !********POSITIONER MOVE******** ;
1252:J P[319] 85% CNT30    ;
1253:   ;
1254:J P[320] 50% CNT25    ;
1255:   ;
1256:L P[321] 1000mm/sec CNT60    ;
1257:   ;
1258:   ;
1259:  !FR50M1510 ;
1260:  IF R[15]=1511,CALL TECH_HOLD ;
1261:   ;
1262:   ;
1263:   ;
1264:L P[389] 1000mm/sec FINE
    :  Arc Start[6]    ;
1265:  Weave Sine[6] ;
1266:  Track TAST[6] ;
1267:L P[392] WELD_SPEED CNT100    ;
1268:L P[393] WELD_SPEED CNT100    ;
1269:L P[394] WELD_SPEED CNT100    ;
1270:L P[395] WELD_SPEED CNT100    ;
1271:L P[396] WELD_SPEED CNT100    ;
1272:L P[397] WELD_SPEED CNT100    ;
1273:L P[398] WELD_SPEED FINE
    :  Arc End[6]    ;
1274:  Weave End ;
1275:  Track End ;
1276:   ;
1277:   ;
1278:L P[328] 1000mm/sec CNT90    ;
1279:   ;
1280:L P[329] 1000mm/sec CNT30    ;
1281:   ;
1282:   ;
1283:  !FR50M1520 ;
1284:  IF R[15]=1521,CALL TECH_HOLD ;
1285:   ;
1286:   ;
1287:   ;
1288:L P[403] 1000mm/sec FINE
    :  Arc Start[6]    ;
1289:  Weave Sine[6] ;
1290:  Track TAST[6] ;
1291:L P[404] WELD_SPEED CNT100    ;
1292:L P[405] WELD_SPEED CNT100    ;
1293:L P[406] WELD_SPEED FINE
    :  Arc End[6]    ;
1294:  Weave End ;
1295:  Track End ;
1296:   ;
1297:   ;
1298:L P[334] 1000mm/sec CNT50    ;
1299:   ;
1300:L P[335] 1400mm/sec CNT90    ;
1301:   ;
1302:J P[763] 50% CNT60    ;
1303:   ;
1304:  !********POSITIONER MOVE******** ;
1305:J P[336] 85% CNT40    ;
1306:   ;
1307:J P[337] 50% CNT25    ;
1308:   ;
1309:L P[338] 1000mm/sec CNT25    ;
1310:   ;
1311:   ;
1312:  !FR50M1530 ;
1313:  IF R[15]=1531,CALL TECH_HOLD ;
1314:   ;
1315:   ;
1316:   ;
1317:L P[407] 1000mm/sec FINE
    :  Arc Start[6]    ;
1318:  Weave Sine[6] ;
1319:  Track TAST[6] ;
1320:L P[408] WELD_SPEED CNT100    ;
1321:L P[409] WELD_SPEED CNT100    ;
1322:L P[410] WELD_SPEED CNT100    ;
1323:L P[411] WELD_SPEED CNT100    ;
1324:L P[412] WELD_SPEED CNT100    ;
1325:L P[415] WELD_SPEED CNT100    ;
1326:L P[416] WELD_SPEED FINE
    :  Arc End[6]    ;
1327:  Weave End ;
1328:  Track End ;
1329:   ;
1330:   ;
1331:L P[344] 1000mm/sec CNT60    ;
1332:   ;
1333:L P[345] 1000mm/sec CNT80    ;
1334:   ;
1335:   ;
1336:  !FR50M1540 ;
1337:  IF R[15]=1541,CALL TECH_HOLD ;
1338:   ;
1339:   ;
1340:   ;
1341:L P[417] 1000mm/sec FINE
    :  Arc Start[6]    ;
1342:  Weave Sine[6] ;
1343:  Track TAST[6] ;
1344:L P[418] WELD_SPEED CNT100    ;
1345:L P[419] WELD_SPEED CNT100    ;
1346:L P[420] WELD_SPEED FINE
    :  Arc End[6]    ;
1347:  Weave End ;
1348:  Track End ;
1349:   ;
1350:   ;
1351:L P[350] 1000mm/sec CNT40    ;
1352:   ;
1353:L P[351] 1000mm/sec CNT25    ;
1354:   ;
1355:  !HOME ;
1356:J P[764] 100% CNT50    ;
1357:   ;
1358:  !********POSITIONER MOVE******** ;
1359:J P[352] 85% CNT70    ;
1360:   ;
1361:  CALL HOME    ;
1362:  CALL T_CLEAN    ;
1363:   ;
1364:J P[353] 50% CNT35    ;
1365:   ;
1366:L P[354] 1000mm/sec CNT40    ;
1367:   ;
1368:  !FR50M1550 ;
1369:  IF R[15]=1551,CALL TECH_HOLD ;
1370:   ;
1371:   ;
1372:   ;
1373:L P[427] 1000mm/sec FINE
    :  Arc Start[6]    ;
1374:  Weave Sine[6] ;
1375:  Track TAST[6] ;
1376:L P[428] WELD_SPEED FINE
    :  Arc End[6]    ;
1377:  Weave End ;
1378:  Track End ;
1379:   ;
1380:   ;
1381:L P[357] 1000mm/sec CNT25    ;
1382:   ;
1383:J P[358] 50% CNT25    ;
1384:   ;
1385:   ;
1386:  !FR50M1560 ;
1387:  IF R[15]=1561,CALL TECH_HOLD ;
1388:   ;
1389:   ;
1390:   ;
1391:L P[433] 1000mm/sec FINE
    :  Arc Start[6]    ;
1392:  Weave Sine[6] ;
1393:  Track TAST[6] ;
1394:L P[434] WELD_SPEED FINE
    :  Arc End[6]    ;
1395:  Weave End ;
1396:  Track End ;
1397:   ;
1398:   ;
1399:L P[361] 1000mm/sec CNT25    ;
1400:   ;
1401:L P[362] 960mm/sec CNT100    ;
1402:   ;
1403:L P[364] 1500mm/sec CNT25    ;
1404:   ;
1405:  !********POSITIONER MOVE******** ;
1406:J P[365] 85% CNT20    ;
1407:   ;
1408:L P[366] 1000mm/sec CNT25    ;
1409:   ;
1410:L P[367] 1000mm/sec CNT35    ;
1411:   ;
1412:L P[699] 1000mm/sec CNT25    ;
1413:   ;
1414:   ;
1415:  !FR50M1570 ;
1416:  IF R[15]=1571,CALL TECH_HOLD ;
1417:   ;
1418:   ;
1419:   ;
1420:L P[441] 1000mm/sec FINE
    :  Arc Start[6]    ;
1421:  Weave Sine[6] ;
1422:  Track TAST[6] ;
1423:L P[442] WELD_SPEED CNT100    ;
1424:L P[445] WELD_SPEED FINE
    :  Arc End[6]    ;
1425:  Weave End ;
1426:  Track End ;
1427:   ;
1428:   ;
1429:L P[371] 1000mm/sec CNT25    ;
1430:   ;
1431:L P[372] 1000mm/sec CNT100    ;
1432:   ;
1433:L P[373] 1000mm/sec CNT100    ;
1434:   ;
1435:L P[374] 1000mm/sec CNT100    ;
1436:   ;
1437:   ;
1438:  !FR50M1580 ;
1439:  IF R[15]=1581,CALL TECH_HOLD ;
1440:   ;
1441:   ;
1442:   ;
1443:L P[446] 1000mm/sec FINE
    :  Arc Start[6]    ;
1444:  Weave Sine[6] ;
1445:  Track TAST[6] ;
1446:L P[450] WELD_SPEED CNT100    ;
1447:L P[451] WELD_SPEED FINE
    :  Arc End[6]    ;
1448:  Weave End ;
1449:  Track End ;
1450:   ;
1451:   ;
1452:L P[377] 1000mm/sec CNT25    ;
1453:   ;
1454:L P[378] 1400mm/sec CNT100    ;
1455:   ;
1456:J P[766] 50% CNT35    ;
1457:   ;
1458:  !********POSITIONER MOVE******** ;
1459:J P[379] 90% CNT30    ;
1460:   ;
1461:L P[380] 1000mm/sec CNT30    ;
1462:   ;
1463:L P[381] 1000mm/sec CNT60    ;
1464:   ;
1465:   ;
1466:  !FR50M1590 ;
1467:  IF R[15]=1591,CALL TECH_HOLD ;
1468:   ;
1469:   ;
1470:   ;
1471:L P[452] 1000mm/sec FINE
    :  Arc Start[6]    ;
1472:  Weave Sine[6] ;
1473:  Track TAST[6] ;
1474:L P[453] WELD_SPEED CNT100    ;
1475:C P[454]
    :  P[455] WELD_SPEED CNT100    ;
1476:L P[456] WELD_SPEED CNT100    ;
1477:L P[457] WELD_SPEED CNT100    ;
1478:L P[458] WELD_SPEED CNT100    ;
1479:L P[459] WELD_SPEED FINE
    :  Arc End[6]    ;
1480:  Weave End ;
1481:  Track End ;
1482:   ;
1483:   ;
1484:L P[390] 1000mm/sec CNT25    ;
1485:   ;
1486:J P[391] 50% CNT25    ;
1487:   ;
1488:  !FR50M1600 ;
1489:  IF R[15]=1601,CALL TECH_HOLD ;
1490:   ;
1491:L P[462] 1000mm/sec FINE
    :  Arc Start[6]    ;
1492:  Weave Sine[6] ;
1493:  Track TAST[6] ;
1494:L P[463] WELD_SPEED CNT100    ;
1495:C P[467]
    :  P[468] WELD_SPEED CNT100    ;
1496:L P[471] WELD_SPEED CNT100    ;
1497:C P[472]
    :  P[477] WELD_SPEED CNT100    ;
1498:L P[478] WELD_SPEED FINE
    :  Arc End[6]    ;
1499:  Weave End ;
1500:  Track End ;
1501:   ;
1502:   ;
1503:L P[399] 1000mm/sec CNT35    ;
1504:   ;
1505:  !********POSITIONER MOVE******** ;
1506:J P[400] 85% CNT30    ;
1507:   ;
1508:J P[401] 50% CNT35    ;
1509:   ;
1510:L P[402] 1000mm/sec CNT40    ;
1511:   ;
1512:L P[702] 1000mm/sec CNT30    ;
1513:   ;
1514:   ;
1515:  !FR50M1610 ;
1516:  IF R[15]=1611,CALL TECH_HOLD ;
1517:   ;
1518:   ;
1519:   ;
1520:L P[95] 1000mm/sec FINE
    :  Arc Start[6]    ;
1521:  Weave Sine[6] ;
1522:  Track TAST[6] ;
1523:L P[97] WELD_SPEED CNT100    ;
1524:C P[100]
    :  P[101] WELD_SPEED CNT100    ;
1525:L P[104] WELD_SPEED CNT100    ;
1526:L P[105] WELD_SPEED FINE
    :  Arc End[6]    ;
1527:  Track End ;
1528:  Weave End ;
1529:   ;
1530:L P[704] 800mm/sec CNT25    ;
1531:   ;
1532:L P[705] 800mm/sec CNT10    ;
1533:   ;
1534:L P[706] 800mm/sec CNT10    ;
1535:   ;
1536:   ;
1537:  !FR50M1610 continued ;
1538:  IF R[15]=1611,CALL TECH_HOLD ;
1539:   ;
1540:   ;
1541:L P[106] 800mm/sec FINE
    :  Arc Start[6]    ;
1542:  Weave Sine[6] ;
1543:  Track TAST[6] ;
1544:L P[107] WELD_SPEED CNT100    ;
1545:L P[112] WELD_SPEED CNT100    ;
1546:C P[113]
    :  P[114] WELD_SPEED CNT100    ;
1547:C P[115]
    :  P[119] WELD_SPEED CNT100    ;
1548:L P[120] WELD_SPEED FINE
    :  Arc End[6]    ;
1549:  Weave End ;
1550:  Track End ;
1551:   ;
1552:L P[413] 1000mm/sec CNT100    ;
1553:   ;
1554:L P[414] 1000mm/sec CNT100    ;
1555:   ;
1556:   ;
1557:  !FR50M1611 CONTINUED ;
1558:  IF R[15]=1612,CALL TECH_HOLD ;
1559:   ;
1560:   ;
1561:   ;
1562:L P[514] 1000mm/sec FINE
    :  Arc Start[6]    ;
1563:  Weave Sine[6] ;
1564:  Track TAST[6] ;
1565:L P[515] WELD_SPEED CNT100    ;
1566:C P[517]
    :  P[518] WELD_SPEED CNT100    ;
1567:C P[520]
    :  P[521] WELD_SPEED FINE
    :  Arc End[6]    ;
1568:  Weave End ;
1569:  Track End ;
1570:   ;
1571:   ;
1572:L P[421] 1000mm/sec CNT80    ;
1573:   ;
1574:L P[422] 1400mm/sec CNT50    ;
1575:   ;
1576:J P[668] 50% CNT30    ;
1577:   ;
1578:  !********POSITIONER MOVE******** ;
1579:J P[424] 85% CNT30    ;
1580:   ;
1581:J P[669] 50% CNT70    ;
1582:   ;
1583:J P[426] 40% CNT25    ;
1584:   ;
1585:   ;
1586:  !FR50M1630 ;
1587:  IF R[15]=1631,CALL TECH_HOLD ;
1588:   ;
1589:   ;
1590:   ;
1591:L P[522] 1000mm/sec FINE
    :  Arc Start[6]    ;
1592:  Weave Sine[6] ;
1593:  Track TAST[6] ;
1594:L P[526] WELD_SPEED FINE
    :  Arc End[6]    ;
1595:  Weave End ;
1596:  Track End ;
1597:   ;
1598:   ;
1599:L P[429] 1000mm/sec CNT25    ;
1600:   ;
1601:J P[430] 50% CNT25    ;
1602:   ;
1603:L P[431] 1000mm/sec CNT25    ;
1604:   ;
1605:L P[432] 1000mm/sec CNT25    ;
1606:   ;
1607:   ;
1608:  !FR50M1640 ;
1609:  IF R[15]=1641,CALL TECH_HOLD ;
1610:   ;
1611:   ;
1612:   ;
1613:L P[527] 500mm/sec FINE
    :  Arc Start[6]    ;
1614:  Weave Sine[6] ;
1615:  Track TAST[6] ;
1616:L P[532] WELD_SPEED FINE
    :  Arc End[6]    ;
1617:  Weave End ;
1618:  Track End ;
1619:   ;
1620:   ;
1621:L P[435] 1000mm/sec CNT25    ;
1622:   ;
1623:L P[436] 1000mm/sec CNT25    ;
1624:   ;
1625:L P[437] 1000mm/sec CNT30    ;
1626:   ;
1627:  !********POSITIONER MOVE******** ;
1628:J P[438] 70% CNT30    ;
1629:   ;
1630:L P[712] 1000mm/sec CNT30    ;
1631:   ;
1632:L P[439] 1000mm/sec CNT25    ;
1633:   ;
1634:L P[440] 1000mm/sec CNT25    ;
1635:   ;
1636:   ;
1637:  !FR50M1650 ;
1638:  IF R[15]=1651,CALL TECH_HOLD ;
1639:   ;
1640:   ;
1641:   ;
1642:L P[533] 1000mm/sec FINE
    :  Arc Start[6]    ;
1643:  Weave Sine[6] ;
1644:  Track TAST[6] ;
1645:L P[534] WELD_SPEED CNT100    ;
1646:L P[535] WELD_SPEED CNT100    ;
1647:L P[536] WELD_SPEED FINE
    :  Arc End[6]    ;
1648:  Weave End ;
1649:  Track End ;
1650:   ;
1651:   ;
1652:L P[443] 300mm/sec CNT25    ;
1653:   ;
1654:L P[713] 300mm/sec CNT5    ;
1655:   ;
1656:L P[714] 800mm/sec CNT5    ;
1657:   ;
1658:  !********POSITIONER MOVE******** ;
1659:J P[444] 80% CNT10    ;
1660:   ;
1661:   ;
1662:  !FR50M1660 ;
1663:  IF R[15]=1661,CALL TECH_HOLD ;
1664:   ;
1665:   ;
1666:   ;
1667:L P[537] 100mm/sec FINE
    :  Arc Start[6]    ;
1668:  Weave Sine[6] ;
1669:  Track TAST[6] ;
1670:L P[540] WELD_SPEED CNT100    ;
1671:L P[541] WELD_SPEED FINE
    :  Arc End[6]    ;
1672:  Weave End ;
1673:  Track End ;
1674:   ;
1675:   ;
1676:L P[447] 300mm/sec CNT25    ;
1677:   ;
1678:L P[448] 500mm/sec CNT30    ;
1679:   ;
1680:L P[449] 1000mm/sec CNT40    ;
1681:   ;
1682:   ;
1683:  !FR50M1670 ;
1684:  IF R[15]=1671,CALL TECH_HOLD ;
1685:   ;
1686:   ;
1687:   ;
1688:L P[542] 1000mm/sec FINE
    :  Arc Start[6]    ;
1689:  Weave Sine[6] ;
1690:  Track TAST[6] ;
1691:L P[543] WELD_SPEED CNT100    ;
1692:C P[544]
    :  P[545] WELD_SPEED CNT100    ;
1693:L P[546] WELD_SPEED CNT100    ;
1694:C P[550]
    :  P[551] 16.0inch/min CNT100    ;
1695:L P[552] WELD_SPEED CNT100    ;
1696:C P[555]
    :  P[556] WELD_SPEED FINE
    :  Arc End[6]    ;
1697:  Weave End ;
1698:  Track End ;
1699:   ;
1700:   ;
1701:L P[460] 1000mm/sec CNT30    ;
1702:   ;
1703:L P[461] 1000mm/sec CNT40    ;
1704:   ;
1705:   ;
1706:  !FR50M1680 ;
1707:  IF R[15]=1681,CALL TECH_HOLD ;
1708:   ;
1709:   ;
1710:   ;
1711:L P[558] 1000mm/sec FINE
    :  Arc Start[6]    ;
1712:  Weave Sine[6] ;
1713:  Track TAST[6] ;
1714:L P[559] WELD_SPEED CNT100    ;
1715:L P[561] WELD_SPEED FINE
    :  Arc End[6]    ;
1716:  Weave End ;
1717:  Track End ;
1718:   ;
1719:   ;
1720:L P[464] 1000mm/sec CNT25    ;
1721:   ;
1722:  !********POSITIONER MOVE******** ;
1723:J P[465] 75% CNT10    ;
1724:   ;
1725:L P[466] 1000mm/sec CNT25    ;
1726:   ;
1727:   ;
1728:  !FR50M1690 ;
1729:  IF R[15]=1691,CALL TECH_HOLD ;
1730:   ;
1731:   ;
1732:   ;
1733:L P[562] 1000mm/sec FINE
    :  Arc Start[8]    ;
1734:  Weave Sine[8] ;
1735:L P[564] WELD_SPEED FINE
    :  Arc End[8]    ;
1736:  Weave End ;
1737:   ;
1738:   ;
1739:L P[469] 1000mm/sec CNT40    ;
1740:   ;
1741:L P[470] 1000mm/sec CNT40    ;
1742:   ;
1743:   ;
1744:  !FR50M11700 ;
1745:  IF R[15]=1171,CALL TECH_HOLD ;
1746:   ;
1747:   ;
1748:L P[123] 1000mm/sec FINE
    :  Arc Start[6]    ;
1749:  Weave Sine[6] ;
1750:  Track TAST[6] ;
1751:L P[343] WELD_SPEED FINE
    :  Arc End[6]    ;
1752:  Weave End ;
1753:  Track End ;
1754:   ;
1755:L P[473] 1000mm/sec CNT50    ;
1756:   ;
1757:L P[673] 1000mm/sec CNT70    ;
1758:   ;
1759:J P[474] 50% CNT25    ;
1760:   ;
1761:  !********POSITIONER MOVE******** ;
1762:J P[475] 85% CNT15    ;
1763:   ;
1764:L P[476] 1000mm/sec CNT25    ;
1765:   ;
1766:   ;
1767:  !FR50M1710 ;
1768:  IF R[15]=1711,CALL TECH_HOLD ;
1769:   ;
1770:   ;
1771:   ;
1772:L P[572] 1000mm/sec FINE
    :  Arc Start[6]    ;
1773:  Weave Sine[6] ;
1774:  Track TAST[6] ;
1775:L P[573] WELD_SPEED CNT100    ;
1776:L P[574] WELD_SPEED FINE
    :  Arc End[6]    ;
1777:  Weave End ;
1778:  Track End ;
1779:   ;
1780:   ;
1781:L P[479] 1000mm/sec CNT35    ;
1782:   ;
1783:   ;
1784:  !FR50M1720 ;
1785:  IF R[15]=1721,CALL TECH_HOLD ;
1786:   ;
1787:   ;
1788:L P[575] 1000mm/sec FINE
    :  Arc Start[6]    ;
1789:  Weave Sine[6] ;
1790:L P[577] WELD_SPEED CNT100    ;
1791:L P[578] WELD_SPEED CNT100    ;
1792:L P[579] WELD_SPEED FINE
    :  Arc End[6]    ;
1793:  Weave End ;
1794:   ;
1795:   ;
1796:L P[484] 1000mm/sec CNT35    ;
1797:   ;
1798:L P[485] 1000mm/sec CNT50    ;
1799:   ;
1800:   ;
1801:  !FR50M1730 ;
1802:  IF R[15]=1731,CALL TECH_HOLD ;
1803:   ;
1804:   ;
1805:   ;
1806:L P[580] 1000mm/sec FINE
    :  Arc Start[6]    ;
1807:  Weave Sine[6] ;
1808:  Track TAST[6] ;
1809:L P[581] WELD_SPEED FINE
    :  Arc End[6]    ;
1810:  Weave End ;
1811:  Track End ;
1812:   ;
1813:   ;
1814:L P[488] 1000mm/sec CNT25    ;
1815:   ;
1816:L P[489] 1000mm/sec CNT25    ;
1817:   ;
1818:   ;
1819:  !FR50M1740 ;
1820:  IF R[15]=1741,CALL TECH_HOLD ;
1821:   ;
1822:   ;
1823:   ;
1824:L P[582] 1000mm/sec FINE
    :  Arc Start[6]    ;
1825:  Weave Sine[6] ;
1826:  Track TAST[6] ;
1827:L P[583] WELD_SPEED CNT100    ;
1828:L P[584] WELD_SPEED FINE
    :  Arc End[6]    ;
1829:  Weave End ;
1830:  Track End ;
1831:   ;
1832:   ;
1833:L P[492] 1000mm/sec CNT25    ;
1834:   ;
1835:L P[493] 1000mm/sec CNT50    ;
1836:   ;
1837:L P[494] 1000mm/sec CNT25    ;
1838:   ;
1839:L P[495] 1500mm/sec CNT70    ;
1840:   ;
1841:J P[496] 50% CNT30    ;
1842:   ;
1843:   ;
1844:  !FR50M1750 ;
1845:  IF R[15]=1751,CALL TECH_HOLD ;
1846:   ;
1847:   ;
1848:L P[497] 1000mm/sec CNT60    ;
1849:   ;
1850:   ;
1851:L P[585] 1000mm/sec FINE
    :  Arc Start[6]    ;
1852:  Weave Sine[6] ;
1853:  Track TAST[6] ;
1854:L P[586] WELD_SPEED FINE
    :  Arc End[6]    ;
1855:  Weave End ;
1856:  Track End ;
1857:   ;
1858:   ;
1859:L P[500] 1000mm/sec CNT25    ;
1860:   ;
1861:   ;
1862:  !FR50M1760 ;
1863:  IF R[15]=1761,CALL TECH_HOLD ;
1864:   ;
1865:   ;
1866:J P[501] 50% CNT25    ;
1867:   ;
1868:   ;
1869:L P[587] 1000mm/sec FINE
    :  Arc Start[6]    ;
1870:  Weave Sine[6] ;
1871:  Track TAST[6] ;
1872:L P[588] WELD_SPEED FINE
    :  Arc End[6]    ;
1873:  Weave End ;
1874:  Track End ;
1875:   ;
1876:   ;
1877:L P[504] 1000mm/sec CNT30    ;
1878:   ;
1879:L P[505] 1500mm/sec CNT80    ;
1880:   ;
1881:  !********POSITIONER MOVE******** ;
1882:J P[506] 85% CNT50    ;
1883:   ;
1884:J P[507] 50% CNT25    ;
1885:   ;
1886:L P[508] 1000mm/sec CNT25    ;
1887:   ;
1888:L P[509] 1000mm/sec CNT25    ;
1889:   ;
1890:   ;
1891:  !FR50M1770 ;
1892:  IF R[15]=1771,CALL TECH_HOLD ;
1893:   ;
1894:   ;
1895:   ;
1896:L P[590] 1000mm/sec FINE
    :  Arc Start[6]    ;
1897:  Weave Sine[6] ;
1898:  Track TAST[6] ;
1899:L P[591] WELD_SPEED FINE
    :  Arc End[6]    ;
1900:  Weave End ;
1901:  Track End ;
1902:   ;
1903:   ;
1904:L P[512] 1000mm/sec CNT25    ;
1905:   ;
1906:  !********POSITIONER MOVE******** ;
1907:J P[513] 75% CNT20    ;
1908:   ;
1909:   ;
1910:  !FR50M1780 ;
1911:  IF R[15]=1781,CALL TECH_HOLD ;
1912:   ;
1913:   ;
1914:   ;
1915:L P[592] 1000mm/sec FINE
    :  Arc Start[6]    ;
1916:  Weave Sine[6] ;
1917:  Track TAST[6] ;
1918:L P[593] WELD_SPEED FINE
    :  Arc End[6]    ;
1919:  Weave End ;
1920:  Track End ;
1921:   ;
1922:   ;
1923:L P[516] 500mm/sec CNT25    ;
1924:   ;
1925:   ;
1926:  !FR50M1790 ;
1927:  IF R[15]=1791,CALL TECH_HOLD ;
1928:   ;
1929:   ;
1930:   ;
1931:L P[594] 1000mm/sec FINE
    :  Arc Start[6]    ;
1932:  Weave Sine[6] ;
1933:  Track TAST[6] ;
1934:L P[595] WELD_SPEED CNT100    ;
1935:L P[596] WELD_SPEED FINE
    :  Arc End[6]    ;
1936:  Weave End ;
1937:  Track End ;
1938:   ;
1939:   ;
1940:L P[519] 1000mm/sec CNT25    ;
1941:   ;
1942:   ;
1943:  !FR50M1800 ;
1944:  IF R[15]=1801,CALL TECH_HOLD ;
1945:   ;
1946:   ;
1947:   ;
1948:L P[597] 1000mm/sec FINE
    :  Arc Start[6]    ;
1949:  Weave Sine[6] ;
1950:  Track TAST[6] ;
1951:L P[598] WELD_SPEED CNT100    ;
1952:L P[605] WELD_SPEED FINE
    :  Arc End[6]    ;
1953:  Weave End ;
1954:  Track End ;
1955:   ;
1956:   ;
1957:L P[523] 1000mm/sec CNT40    ;
1958:   ;
1959:J P[524] 50% CNT25    ;
1960:   ;
1961:L P[525] 1000mm/sec CNT25    ;
1962:   ;
1963:   ;
1964:  !FR50M1810 ;
1965:  IF R[15]=1811,CALL TECH_HOLD ;
1966:   ;
1967:L P[606] 1000mm/sec FINE
    :  Arc Start[6]    ;
1968:  Weave Sine[6] ;
1969:  Track TAST[6] ;
1970:L P[607] WELD_SPEED CNT100    ;
1971:L P[608] WELD_SPEED FINE
    :  Arc End[6]    ;
1972:  Weave End ;
1973:  Track End ;
1974:   ;
1975:   ;
1976:L P[528] 1000mm/sec CNT25    ;
1977:   ;
1978:J P[529] 60% CNT35    ;
1979:   ;
1980:L P[530] 1500mm/sec CNT60    ;
1981:   ;
1982:L P[531] 1500mm/sec CNT25    ;
1983:   ;
1984:   ;
1985:  !FR50M1820 ;
1986:  IF R[15]=1821,CALL TECH_HOLD ;
1987:   ;
1988:   ;
1989:   ;
1990:L P[609] 1000mm/sec FINE
    :  Arc Start[6]    ;
1991:  Weave Sine[6] ;
1992:  Track TAST[6] ;
1993:L P[610] WELD_SPEED CNT100    ;
1994:C P[611]
    :  P[612] WELD_SPEED CNT100    ;
1995:L P[618] WELD_SPEED CNT100    ;
1996:L P[619] WELD_SPEED FINE
    :  Arc End[6]    ;
1997:  Weave End ;
1998:  Track End ;
1999:   ;
2000:   ;
2001:L P[538] 1000mm/sec CNT30    ;
2002:   ;
2003:J P[539] 50% CNT25    ;
2004:   ;
2005:   ;
2006:  !FR50M1830 ;
2007:  IF R[15]=1831,CALL TECH_HOLD ;
2008:   ;
2009:   ;
2010:   ;
2011:L P[622] 1000mm/sec FINE
    :  Arc Start[6]    ;
2012:  Weave Sine[6] ;
2013:  Track TAST[6] ;
2014:L P[623] WELD_SPEED CNT100    ;
2015:C P[626]
    :  P[627] WELD_SPEED CNT100    ;
2016:L P[629] WELD_SPEED CNT100    ;
2017:C P[630]
    :  P[633] WELD_SPEED CNT100    ;
2018:L P[637] WELD_SPEED FINE
    :  Arc End[6]    ;
2019:  Weave End ;
2020:  Track End ;
2021:   ;
2022:   ;
2023:L P[722] 1000mm/sec CNT60    ;
2024:   ;
2025:L P[547] 1000mm/sec CNT40    ;
2026:   ;
2027:J P[670] 100% CNT50    ;
2028:   ;
2029:J P[548] 60% CNT40    ;
2030:   ;
2031:L P[549] 1000mm/sec CNT30    ;
2032:   ;
2033:L P[723] 1000mm/sec CNT40    ;
2034:   ;
2035:   ;
2036:  !FR50M1840 ;
2037:  IF R[15]=1841,CALL TECH_HOLD ;
2038:   ;
2039:   ;
2040:   ;
2041:L P[638] 1000mm/sec FINE
    :  Arc Start[6]    ;
2042:  Weave Sine[6] ;
2043:L P[639] WELD_SPEED CNT100    ;
2044:L P[640] WELD_SPEED CNT100    ;
2045:L P[641] WELD_SPEED FINE
    :  Arc End[6]    ;
2046:  Weave End ;
2047:   ;
2048:   ;
2049:L P[553] 1000mm/sec CNT25    ;
2050:   ;
2051:L P[554] 1000mm/sec CNT50    ;
2052:   ;
2053:   ;
2054:  !FR50M1850 ;
2055:  IF R[15]=1851,CALL TECH_HOLD ;
2056:   ;
2057:   ;
2058:   ;
2059:L P[642] 1000mm/sec FINE
    :  Arc Start[6]    ;
2060:  Weave Sine[6] ;
2061:  Track TAST[6] ;
2062:L P[647] WELD_SPEED FINE
    :  Arc End[6]    ;
2063:  Weave End ;
2064:  Track End ;
2065:   ;
2066:   ;
2067:L P[557] 1000mm/sec CNT25    ;
2068:   ;
2069:   ;
2070:  !FR50M1860 ;
2071:  IF R[15]=1861,CALL TECH_HOLD ;
2072:   ;
2073:   ;
2074:L P[648] 1000mm/sec FINE
    :  Arc Start[6]    ;
2075:  Weave Sine[6] ;
2076:  Track TAST[6] ;
2077:L P[649] WELD_SPEED CNT100    ;
2078:L P[650] WELD_SPEED FINE
    :  Arc End[6]    ;
2079:  Weave End ;
2080:  Track End ;
2081:   ;
2082:   ;
2083:L P[560] 1000mm/sec CNT25    ;
2084:   ;
2085:   ;
2086:  !FR50M1870 ;
2087:  IF R[15]=1871,CALL TECH_HOLD ;
2088:   ;
2089:   ;
2090:   ;
2091:L P[658] 1000mm/sec FINE
    :  Arc Start[6]    ;
2092:  Weave Sine[6] ;
2093:  Track TAST[6] ;
2094:L P[659] WELD_SPEED CNT100    ;
2095:L P[660] WELD_SPEED FINE
    :  Arc End[6]    ;
2096:  Weave End ;
2097:  Track End ;
2098:   ;
2099:   ;
2100:J P[563] 75% CNT10    ;
2101:   ;
2102:J P[566] 75% CNT10    ;
2103:   ;
2104:   ;
2105:  !FR50M1880 ;
2106:  IF R[15]=1881,CALL TECH_HOLD ;
2107:   ;
2108:   ;
2109:   ;
2110:L P[661] 1000mm/sec FINE
    :  Arc Start[6]    ;
2111:  Weave Sine[6] ;
2112:  Track TAST[6] ;
2113:L P[674] WELD_SPEED FINE
    :  Arc End[6]    ;
2114:  Weave End ;
2115:  Track End ;
2116:   ;
2117:   ;
2118:L P[569] 1000mm/sec CNT25    ;
2119:   ;
2120:  !********POSITIONER MOVE******** ;
2121:J P[570] 75% CNT15    ;
2122:   ;
2123:   ;
2124:  !FR50M1890 ;
2125:  IF R[15]=1891,CALL TECH_HOLD ;
2126:   ;
2127:   ;
2128:L P[571] 1000mm/sec CNT35    ;
2129:   ;
2130:L P[346] 1000mm/sec FINE
    :  Arc Start[6]    ;
2131:  Weave Sine[6] ;
2132:  Track TAST[6] ;
2133:L P[347] WELD_SPEED CNT100    ;
2134:C P[348]
    :  P[349] WELD_SPEED CNT100    ;
2135:L P[355] WELD_SPEED CNT100    ;
2136:L P[490] WELD_SPEED CNT100    ;
2137:L P[491] WELD_SPEED FINE
    :  Arc End[6]    ;
2138:  Track End ;
2139:  Weave End ;
2140:   ;
2141:   ;
2142:L P[730] 800mm/sec CNT30    ;
2143:   ;
2144:L P[731] 800mm/sec CNT25    ;
2145:   ;
2146:L P[732] 800mm/sec CNT30    ;
2147:   ;
2148:   ;
2149:  !FR50M1890 continued ;
2150:  IF R[15]=1891,CALL TECH_HOLD ;
2151:   ;
2152:   ;
2153:L P[498] 800mm/sec FINE
    :  Arc Start[6]    ;
2154:  Weave Sine[6] ;
2155:  Track TAST[6] ;
2156:L P[499] WELD_SPEED CNT100    ;
2157:L P[502] WELD_SPEED CNT100    ;
2158:L P[503] WELD_SPEED CNT100    ;
2159:C P[510]
    :  P[511] WELD_SPEED CNT100    ;
2160:L P[567] WELD_SPEED CNT100    ;
2161:C P[568]
    :  P[682] WELD_SPEED CNT100    ;
2162:C P[683]
    :  P[684] WELD_SPEED CNT100    ;
2163:L P[686] WELD_SPEED FINE
    :  Arc End[6]    ;
2164:  Weave End ;
2165:  Track End ;
2166:   ;
2167:L P[589] 1000mm/sec CNT90    ;
2168:   ;
2169:   ;
2170:  !FR50M1891 ;
2171:  IF R[15]=1892,CALL TECH_HOLD ;
2172:   ;
2173:   ;
2174:   ;
2175:L P[698] 1000mm/sec FINE
    :  Arc Start[6]    ;
2176:  Weave Sine[6] ;
2177:  Track TAST[6] ;
2178:L P[700] WELD_SPEED CNT100    ;
2179:C P[701]
    :  P[703] WELD_SPEED CNT100    ;
2180:L P[707] WELD_SPEED CNT100    ;
2181:C P[708]
    :  P[709] WELD_SPEED CNT100    ;
2182:L P[710] WELD_SPEED CNT100    ;
2183:L P[711] WELD_SPEED FINE
    :  Arc End[6]    ;
2184:  Weave End ;
2185:  Track End ;
2186:   ;
2187:   ;
2188:L P[599] 1000mm/sec CNT25    ;
2189:   ;
2190:L P[600] 1000mm/sec CNT100    ;
2191:   ;
2192:L P[601] 1200mm/sec CNT25    ;
2193:   ;
2194:J P[671] 50% CNT40    ;
2195:   ;
2196:J P[602] 55% CNT25    ;
2197:   ;
2198:  !********POSITIONER MOVE******** ;
2199:J P[603] 85% CNT25    ;
2200:   ;
2201:   ;
2202:  !FR50M1900 ;
2203:  IF R[15]=1901,CALL TECH_HOLD ;
2204:   ;
2205:  CALL ARC_LH_DISABLE_LS(0) ;
2206:   ;
2207:L P[604] 1500mm/sec CNT40    ;
2208:   ;
2209:   ;
2210:L P[715] 1000mm/sec FINE
    :  Arc Start[8]    ;
2211:  Weave Sine[8] ;
2212:L P[716] WELD_SPEED CNT100    ;
2213:C P[717]
    :  P[718] WELD_SPEED CNT100    ;
2214:L P[719] WELD_SPEED CNT100    ;
2215:L P[720] WELD_SPEED CNT100    ;
2216:L P[721] WELD_SPEED CNT100    ;
2217:L P[724] WELD_SPEED FINE
    :  Arc End[8]    ;
2218:  Weave End ;
2219:   ;
2220:   ;
2221:  CALL ARC_LH_DISABLE_LS(1) ;
2222:   ;
2223:L P[613] 1000mm/sec CNT25    ;
2224:   ;
2225:J P[614] 50% CNT50    ;
2226:   ;
2227:J P[672] 100% CNT65    ;
2228:   ;
2229:  !HOME ;
2230:J P[769] 100% CNT25    ;
2231:   ;
2232:  CALL HOME    ;
2233:  CALL T_CLEAN    ;
2234:   ;
2235:  !********POSITIONER MOVE******** ;
2236:J P[615] 85% CNT30    ;
2237:   ;
2238:J P[616] 55% CNT40    ;
2239:   ;
2240:L P[617] 1000mm/sec CNT25    ;
2241:   ;
2242:  CALL ARC_DISABLE_FRONT_BMPR_MED(0) ;
2243:   ;
2244:  //UALM[20] ;
2245:  //!REWORK REQUEST ;
2246:   ;
2247:   ;
2248:  !FR50M1910 ;
2249:  IF R[15]=1911,CALL TECH_HOLD ;
2250:   ;
2251:   ;
2252:   ;
2253:L P[725] 1000mm/sec FINE
    :  Arc Start[6]    ;
2254:  Weave Sine[6] ;
2255:  Track TAST[6] ;
2256:L P[726] WELD_SPEED FINE
    :  Arc End[6]    ;
2257:  Weave End ;
2258:  Track End ;
2259:   ;
2260:   ;
2261:L P[620] 1000mm/sec CNT100    ;
2262:   ;
2263:L P[621] 1000mm/sec CNT100    ;
2264:   ;
2265:   ;
2266:  !FR50M1920 ;
2267:  IF R[15]=1921,CALL TECH_HOLD ;
2268:   ;
2269:   ;
2270:   ;
2271:L P[727] 1000mm/sec FINE
    :  Arc Start[6]    ;
2272:  Weave Sine[6] ;
2273:  Track TAST[6] ;
2274:L P[728] WELD_SPEED FINE
    :  Arc End[6]    ;
2275:  Weave End ;
2276:  Track End ;
2277:   ;
2278:   ;
2279:L P[624] 1000mm/sec CNT100    ;
2280:   ;
2281:L P[625] 1000mm/sec CNT100    ;
2282:   ;
2283:   ;
2284:  !FR50M1930 ;
2285:  IF R[15]=1931,CALL TECH_HOLD ;
2286:   ;
2287:   ;
2288:   ;
2289:L P[729] 1000mm/sec FINE
    :  Arc Start[6]    ;
2290:  Weave Sine[6] ;
2291:  Track TAST[6] ;
2292:L P[733] WELD_SPEED FINE
    :  Arc End[6]    ;
2293:  Weave End ;
2294:  Track End ;
2295:   ;
2296:   ;
2297:  CALL ARC_DISABLE_FRONT_BMPR_MED(1) ;
2298:   ;
2299:   ;
2300:L P[628] 1000mm/sec CNT100    ;
2301:   ;
2302:J P[771] 70% CNT30    ;
2303:   ;
2304:  !********POSITIONER MOVE******** ;
2305:J P[644] 85% CNT30    ;
2306:   ;
2307:L P[645] 1000mm/sec CNT25    ;
2308:   ;
2309:  CALL ARC_LH_DISABLE_LS(0) ;
2310:   ;
2311:   ;
2312:  !FR50M1960 ;
2313:  IF R[15]=1961,CALL TECH_HOLD ;
2314:   ;
2315:L P[646] 300mm/sec CNT25    ;
2316:   ;
2317:L P[734] 1000mm/sec FINE
    :  Arc Start[6]    ;
2318:  Weave Sine[6] ;
2319:  Track TAST[6] ;
2320:L P[735] WELD_SPEED CNT100    ;
2321:L P[736] WELD_SPEED CNT100    ;
2322:C P[737]
    :  P[738] WELD_SPEED FINE
    :  Arc End[6]    ;
2323:  Weave End ;
2324:  Track End ;
2325:   ;
2326:   ;
2327:L P[651] 1000mm/sec CNT25    ;
2328:   ;
2329:  CALL ARC_LH_DISABLE_LS(1) ;
2330:   ;
2331:L P[652] 1000mm/sec CNT100    ;
2332:   ;
2333:L P[653] 1000mm/sec CNT25    ;
2334:   ;
2335:J P[202] 50% CNT30    ;
2336:   ;
2337:  !********POSITIONER MOVE******** ;
2338:J P[91] 85% CNT40    ;
2339:   ;
2340:J P[423] 75% CNT40    ;
2341:   ;
2342:L P[576] 1000mm/sec CNT80    ;
2343:   ;
2344:  CALL ARC_DISABLE_RH_LS(0) ;
2345:   ;
2346:   ;
2347:  !FR50M1971 ;
2348:  IF R[15]=1972,CALL TECH_HOLD ;
2349:   ;
2350:   ;
2351:   ;
2352:L P[746] 800mm/sec FINE
    :  Arc Start[6]    ;
2353:  Weave Sine[6] ;
2354:  Track TAST[6] ;
2355:L P[747] WELD_SPEED CNT100    ;
2356:C P[751]
    :  P[752] WELD_SPEED FINE
    :  Arc End[6]    ;
2357:  Track End ;
2358:  Weave End ;
2359:   ;
2360:   ;
2361:L P[654] 800mm/sec CNT5    ;
2362:   ;
2363:J P[664] 25% CNT40    ;
2364:   ;
2365:J P[665] 50% CNT25    ;
2366:   ;
2367:J P[666] 75% CNT40    ;
2368:   ;
2369:J P[667] 50% CNT50    ;
2370:   ;
2371:  !********POSITIONER MOVE******** ;
2372:J P[655] 85% CNT30    ;
2373:   ;
2374:J P[656] 55% CNT25    ;
2375:   ;
2376:   ;
2377:  !FR50M1970 ;
2378:  IF R[15]=1971,CALL TECH_HOLD ;
2379:   ;
2380:   ;
2381:L P[657] 1000mm/sec CNT25    ;
2382:   ;
2383:L P[565] 800mm/sec CNT100    ;
2384:   ;
2385:   ;
2386:L P[739] 1000mm/sec FINE
    :  Arc Start[6]    ;
2387:  Weave Sine[6] ;
2388:  Track TAST[6] ;
2389:L P[740] WELD_SPEED CNT100    ;
2390:L P[741] WELD_SPEED CNT100    ;
2391:C P[744]
    :  P[745] WELD_SPEED FINE
    :  Arc End[6]    ;
2392:  Weave End ;
2393:  Track End ;
2394:   ;
2395:   ;
2396:  CALL ARC_DISABLE_RH_LS(1) ;
2397:   ;
2398:L P[662] 500mm/sec CNT25    ;
2399:   ;
2400:L P[663] 1000mm/sec CNT25    ;
2401:   ;
2402:J P[773] 70% CNT40    ;
2403:   ;
2404:  !******** POSITIONER MOVE ******* ;
2405:J P[783] 100% CNT40    ;
2406:   ;
2407:J P[742] 75% CNT35    ;
2408:   ;
2409:L P[743] 1000mm/sec CNT35    ;
2410:   ;
2411:  CALL ARC_LH_DISABLE_LS(0) ;
2412:   ;
2413:   ;
2414:  !FR50M1961 ;
2415:  IF R[15]=1962,CALL TECH_HOLD ;
2416:   ;
2417:   ;
2418:   ;
2419:L P[753] 800mm/sec FINE
    :  Arc Start[6]    ;
2420:  Weave Sine[6] ;
2421:  Track TAST[6] ;
2422:L P[754] WELD_SPEED CNT100    ;
2423:C P[755]
    :  P[758] WELD_SPEED FINE
    :  Arc End[6]    ;
2424:  Track End ;
2425:  Weave End ;
2426:   ;
2427:   ;
2428:  CALL ARC_LH_DISABLE_LS(1) ;
2429:   ;
2430:L P[748] 800mm/sec CNT25    ;
2431:   ;
2432:L P[749] 1000mm/sec CNT100    ;
2433:   ;
2434:L P[750] 1000mm/sec CNT70    ;
2435:   ;
2436:  !HOME ;
2437:J P[774] 100% FINE    ;
2438:   ;
2439:  !********POSITIONER MOVE******** ;
2440:  !LOAD POSITION ;
2441:  CALL HOME    ;
2442:  CALL LOAD_POS    ;
2443:  TIMER[12]=STOP ;
2444:   ;
/POS
P[1]{
   GP1:
	UF : 1, UT : 1,		CONFIG : 'N U T, 0, 0, 0',
	X =  1183.912  mm,	Y = -1389.570  mm,	Z =   968.895  mm,
	W =    19.924 deg,	P =    44.168 deg,	R =  -125.816 deg
   GP2:
	UF : 1, UT : 1,
	J1=     0.000 deg,	J2=   -40.000 deg
};
P[2]{
   GP1:
	UF : 1, UT : 1,		CONFIG : 'N U T, 0, 0, 0',
	X =  1125.641  mm,	Y = -1312.769  mm,	Z =   506.026  mm,
	W =     -.010 deg,	P =    46.626 deg,	R =  -140.083 deg
   GP2:
	UF : 1, UT : 1,
	J1=     0.000 deg,	J2=   -40.000 deg
};
P[3]{
   GP1:
	UF : 1, UT : 1,		CONFIG : 'N U T, 0, 0, 0',
	X =  1237.616  mm,	Y = -1312.769  mm,	Z =   231.881  mm,
	W =     -.010 deg,	P =    46.626 deg,	R =  -140.083 deg
   GP2:
	UF : 1, UT : 1,
	J1=     0.000 deg,	J2=   -40.000 deg
};
P[4]{
   GP1:
	UF : 1, UT : 1,		CONFIG : 'N U T, 0, 0, 0',
	X =  1253.715  mm,	Y = -1258.752  mm,	Z =    71.686  mm,
	W =     -.013 deg,	P =    46.636 deg,	R =  -142.462 deg
   GP2:
	UF : 1, UT : 1,
	J1=     0.000 deg,	J2=   -40.000 deg
};
P[5]{
   GP1:
	UF : 1, UT : 1,		CONFIG : 'N U T, 0, 0, 0',
	X =  1297.402  mm,	Y = -1311.211  mm,	Z =    76.271  mm,
	W =     -.716 deg,	P =    46.671 deg,	R =  -171.143 deg
   GP2:
	UF : 1, UT : 1,
	J1=     -.000 deg,	J2=   -40.000 deg
};
P[6]{
   GP1:
	UF : 1, UT : 1,		CONFIG : 'N U T, 0, 0, 0',
	X =  1235.617  mm,	Y = -1318.769  mm,	Z =   246.881  mm,
	W =     -.010 deg,	P =    46.625 deg,	R =  -163.368 deg
   GP2:
	UF : 1, UT : 1,
	J1=     0.000 deg,	J2=   -40.000 deg
};
P[7]{
   GP1:
	UF : 1, UT : 1,		CONFIG : 'N U T, 0, 0, 0',
	X =   831.467  mm,	Y =  -918.769  mm,	Z =   246.881  mm,
	W =     -.010 deg,	P =    46.625 deg,	R =  -137.059 deg
   GP2:
	UF : 1, UT : 1,
	J1=     0.000 deg,	J2=   -40.000 deg
};
P[8]{
   GP1:
	UF : 1, UT : 1,		CONFIG : 'N U T, 0, 0, 0',
	X =   897.240  mm,	Y =  -831.059  mm,	Z =    70.995  mm,
	W =     1.854 deg,	P =    45.123 deg,	R =  -141.040 deg
   GP2:
	UF : 1, UT : 1,
	J1=     0.000 deg,	J2=   -40.000 deg
};
P[9]{
   GP1:
	UF : 1, UT : 1,		CONFIG : 'N U T, 0, 0, 0',
	X =  1066.495  mm,	Y = -1033.818  mm,	Z =    71.044  mm,
	W =     1.854 deg,	P =    45.124 deg,	R =  -141.040 deg
   GP2:
	UF : 1, UT : 1,
	J1=     0.000 deg,	J2=   -40.000 deg
};
P[10]{
   GP1:
	UF : 1, UT : 1,		CONFIG : 'N U T, 0, 0, 0',
	X =  1165.677  mm,	Y = -1317.151  mm,	Z =   195.424  mm,
	W =     2.049 deg,	P =    44.964 deg,	R =  -137.101 deg
   GP2:
	UF : 1, UT : 1,
	J1=     0.000 deg,	J2=   -40.000 deg
};
P[11]{
   GP1:
	UF : 1, UT : 1,		CONFIG : 'N U T, 0, 0, 0',
	X =   788.632  mm,	Y =  -909.151  mm,	Z =   195.424  mm,
	W =     2.049 deg,	P =    44.964 deg,	R =  -137.101 deg
   GP2:
	UF : 1, UT : 1,
	J1=     0.000 deg,	J2=   -40.000 deg
};
P[12]{
   GP1:
	UF : 1, UT : 1,		CONFIG : 'N U T, 0, 0, 0',
	X =  1231.082  mm,	Y = -1228.554  mm,	Z =    70.371  mm,
	W =     1.854 deg,	P =    45.124 deg,	R =  -141.040 deg
   GP2:
	UF : 1, UT : 1,
	J1=     0.000 deg,	J2=   -40.000 deg
};
P[13]{
   GP1:
	UF : 1, UT : 1,		CONFIG : 'N U T, 0, 0, 0',
	X =   871.790  mm,	Y =  -803.766  mm,	Z =    72.955  mm,
	W =     2.049 deg,	P =    44.963 deg,	R =  -137.102 deg
   GP2:
	UF : 1, UT : 1,
	J1=     0.000 deg,	J2=   -40.000 deg
};
P[14]{
   GP1:
	UF : 1, UT : 1,		CONFIG : 'N U T, 0, 0, 0',
	X =   724.617  mm,	Y =  -938.147  mm,	Z =   287.454  mm,
	W =     2.255 deg,	P =    44.853 deg,	R =  -120.173 deg
   GP2:
	UF : 1, UT : 1,
	J1=     0.000 deg,	J2=   -40.000 deg
};
P[15]{
   GP1:
	UF : 1, UT : 1,		CONFIG : 'N U T, 0, 0, 0',
	X =   918.616  mm,	Y =    -7.769  mm,	Z =  2170.023  mm,
	W =     -.010 deg,	P =   -45.000 deg,	R =     0.000 deg
   GP2:
	UF : 1, UT : 1,
	J1=    90.000 deg,	J2=     0.000 deg
};
P[16]{
   GP1:
	UF : 1, UT : 1,		CONFIG : 'N U T, 0, 0, 0',
	X =  2031.616  mm,	Y =    -7.769  mm,	Z =  1188.167  mm,
	W =     -.010 deg,	P =    38.462 deg,	R =   -90.000 deg
   GP2:
	UF : 1, UT : 1,
	J1=    90.000 deg,	J2=     0.000 deg
};
P[17]{
   GP1:
	UF : 1, UT : 1,		CONFIG : 'N U T, 0, 0, 0',
	X =  2496.616  mm,	Y =   140.231  mm,	Z =   484.166  mm,
	W =    29.850 deg,	P =    25.473 deg,	R =   -36.833 deg
   GP2:
	UF : 1, UT : 1,
	J1=    90.000 deg,	J2=     0.000 deg
};
P[18]{
   GP1:
	UF : 1, UT : 1,		CONFIG : 'N U T, 0, 0, 0',
	X =  2496.616  mm,	Y =   299.231  mm,	Z =   410.165  mm,
	W =    38.288 deg,	P =     3.975 deg,	R =    -5.002 deg
   GP2:
	UF : 1, UT : 1,
	J1=    90.000 deg,	J2=     0.000 deg
};
P[19]{
   GP1:
	UF : 1, UT : 1,		CONFIG : 'N U T, 0, 0, 0',
	X =   827.497  mm,	Y =  -749.395  mm,	Z =    73.174  mm,
	W =     2.121 deg,	P =    44.922 deg,	R =  -125.436 deg
   GP2:
	UF : 1, UT : 1,
	J1=     0.000 deg,	J2=   -40.000 deg
};
P[20]{
   GP1:
	UF : 1, UT : 1,		CONFIG : 'N U T, 0, 0, 0',
	X =  2508.544  mm,	Y =   411.773  mm,	Z =   343.204  mm,
	W =    44.831 deg,	P =     4.520 deg,	R =     -.858 deg
   GP2:
	UF : 1, UT : 1,
	J1=    90.000 deg,	J2=     0.000 deg
};
P[21]{
   GP1:
	UF : 1, UT : 1,		CONFIG : 'N U T, 0, 0, 0',
	X =  2563.389  mm,	Y =   199.190  mm,	Z =   572.868  mm,
	W =    44.821 deg,	P =     4.511 deg,	R =    23.598 deg
   GP2:
	UF : 1, UT : 1,
	J1=    90.000 deg,	J2=     0.000 deg
};
P[22]{
   GP1:
	UF : 1, UT : 1,		CONFIG : 'N U T, 0, 0, 0',
	X =  2120.246  mm,	Y =   303.348  mm,	Z =   455.868  mm,
	W =    32.270 deg,	P =    33.247 deg,	R =    37.053 deg
   GP2:
	UF : 1, UT : 1,
	J1=    90.000 deg,	J2=     0.000 deg
};
P[23]{
   GP1:
	UF : 1, UT : 1,		CONFIG : 'N U T, 0, 0, 0',
	X =  2463.469  mm,	Y =   413.974  mm,	Z =   341.292  mm,
	W =    44.821 deg,	P =     4.515 deg,	R =     -.858 deg
   GP2:
	UF : 1, UT : 1,
	J1=    90.000 deg,	J2=     0.000 deg
};
P[24]{
   GP1:
	UF : 1, UT : 1,		CONFIG : 'N U T, 0, 0, 0',
	X =  2444.293  mm,	Y =   409.807  mm,	Z =   345.410  mm,
	W =    45.505 deg,	P =     6.009 deg,	R =    24.416 deg
   GP2:
	UF : 1, UT : 1,
	J1=    89.999 deg,	J2=     0.000 deg
};
P[25]{
   GP1:
	UF : 1, UT : 1,		CONFIG : 'N U T, 0, 0, 0',
	X =  2090.182  mm,	Y =   379.464  mm,	Z =   444.395  mm,
	W =    34.216 deg,	P =    31.228 deg,	R =    42.244 deg
   GP2:
	UF : 1, UT : 1,
	J1=    90.000 deg,	J2=     0.000 deg
};
P[26]{
   GP1:
	UF : 1, UT : 1,		CONFIG : 'N U T, 0, 0, 0',
	X =  2090.182  mm,	Y =  -337.536  mm,	Z =   444.395  mm,
	W =   -39.673 deg,	P =    23.265 deg,	R =   -63.174 deg
   GP2:
	UF : 1, UT : 1,
	J1=    90.000 deg,	J2=     0.000 deg
};
P[27]{
   GP1:
	UF : 1, UT : 1,		CONFIG : 'N U T, 0, 0, 0',
	X =  2007.570  mm,	Y =   317.185  mm,	Z =   365.466  mm,
	W =    34.218 deg,	P =    31.223 deg,	R =    49.930 deg
   GP2:
	UF : 1, UT : 1,
	J1=    90.000 deg,	J2=     0.000 deg
};
P[28]{
   GP1:
	UF : 1, UT : 1,		CONFIG : 'N U T, 0, 0, 0',
	X =  2008.438  mm,	Y =   396.115  mm,	Z =   365.090  mm,
	W =    34.212 deg,	P =    31.231 deg,	R =    41.673 deg
   GP2:
	UF : 1, UT : 1,
	J1=    90.000 deg,	J2=     0.000 deg
};
P[29]{
   GP1:
	UF : 1, UT : 1,		CONFIG : 'N U T, 0, 0, 0',
	X =  2310.394  mm,	Y =  -277.057  mm,	Z =   689.128  mm,
	W =   -43.030 deg,	P =    14.686 deg,	R =   -51.218 deg
   GP2:
	UF : 1, UT : 1,
	J1=    90.000 deg,	J2=     0.000 deg
};
P[30]{
   GP1:
	UF : 1, UT : 1,		CONFIG : 'N U T, 0, 0, 0',
	X =  2310.394  mm,	Y =     5.943  mm,	Z =   689.127  mm,
	W =     8.920 deg,	P =    44.293 deg,	R =   -85.311 deg
   GP2:
	UF : 1, UT : 1,
	J1=    90.000 deg,	J2=     0.000 deg
};
P[31]{
   GP1:
	UF : 1, UT : 1,		CONFIG : 'N U T, 0, 0, 0',
	X =  2746.395  mm,	Y =     1.943  mm,	Z =  -441.873  mm,
	W =    22.103 deg,	P =    42.731 deg,	R =   -76.212 deg
   GP2:
	UF : 1, UT : 1,
	J1=    90.000 deg,	J2=     0.000 deg
};
P[32]{
   GP1:
	UF : 1, UT : 1,		CONFIG : 'N U T, 0, 0, 0',
	X =  2746.395  mm,	Y =   -73.057  mm,	Z =  -441.873  mm,
	W =    22.103 deg,	P =    42.731 deg,	R =   -76.212 deg
   GP2:
	UF : 1, UT : 1,
	J1=    90.000 deg,	J2=     0.000 deg
};
P[33]{
   GP1:
	UF : 1, UT : 1,		CONFIG : 'N U T, 0, 0, 0',
	X =  2007.015  mm,	Y =  -320.227  mm,	Z =   361.609  mm,
	W =   -39.317 deg,	P =    23.931 deg,	R =   -60.583 deg
   GP2:
	UF : 1, UT : 1,
	J1=    90.000 deg,	J2=     0.000 deg
};
P[34]{
   GP1:
	UF : 1, UT : 1,		CONFIG : 'N U T, 0, 0, 0',
	X =  2007.893  mm,	Y =  -399.787  mm,	Z =   362.621  mm,
	W =   -42.995 deg,	P =    14.795 deg,	R =   -72.419 deg
   GP2:
	UF : 1, UT : 1,
	J1=    90.000 deg,	J2=     0.000 deg
};
P[35]{
   GP1:
	UF : 1, UT : 1,		CONFIG : 'N U T, 0, 0, 0',
	X =  2744.395  mm,	Y =   -87.057  mm,	Z =  -441.873  mm,
	W =    22.103 deg,	P =    42.731 deg,	R =   -76.212 deg
   GP2:
	UF : 1, UT : 1,
	J1=    90.000 deg,	J2=     0.000 deg
};
P[36]{
   GP1:
	UF : 1, UT : 1,		CONFIG : 'N U T, 0, 0, 0',
	X =  2744.394  mm,	Y =    65.467  mm,	Z =  -441.873  mm,
	W =   -23.734 deg,	P =    41.974 deg,	R =    68.142 deg
   GP2:
	UF : 1, UT : 1,
	J1=    90.000 deg,	J2=     0.000 deg
};
P[37]{
   GP1:
	UF : 1, UT : 1,		CONFIG : 'N U T, 0, 0, 0',
	X =  2745.381  mm,	Y =   -55.185  mm,	Z =  -587.693  mm,
	W =    10.080 deg,	P =    44.098 deg,	R =   -75.679 deg
   GP2:
	UF : 1, UT : 1,
	J1=    90.000 deg,	J2=     0.000 deg
};
P[38]{
   GP1:
	UF : 1, UT : 1,		CONFIG : 'N U T, 0, 0, 0',
	X =  2770.065  mm,	Y =   -56.181  mm,	Z =  -586.428  mm,
	W =    10.085 deg,	P =    44.113 deg,	R =   -75.686 deg
   GP2:
	UF : 1, UT : 1,
	J1=    90.000 deg,	J2=     0.000 deg
};
P[39]{
   GP1:
	UF : 1, UT : 1,		CONFIG : 'N U T, 0, 0, 0',
	X =  2744.395  mm,	Y =    65.467  mm,	Z =  -441.873  mm,
	W =   -23.734 deg,	P =    41.974 deg,	R =    68.142 deg
   GP2:
	UF : 1, UT : 1,
	J1=    90.000 deg,	J2=     0.000 deg
};
P[40]{
   GP1:
	UF : 1, UT : 1,		CONFIG : 'N U T, 0, 0, 0',
	X =  2775.566  mm,	Y =    28.292  mm,	Z =  -509.873  mm,
	W =   -17.996 deg,	P =    21.209 deg,	R =   -11.797 deg
   GP2:
	UF : 1, UT : 1,
	J1=    90.000 deg,	J2=     0.000 deg
};
P[41]{
   GP1:
	UF : 1, UT : 1,		CONFIG : 'N U T, 0, 0, 0',
	X =  2745.338  mm,	Y =    53.845  mm,	Z =  -584.045  mm,
	W =   -14.670 deg,	P =    41.217 deg,	R =    68.267 deg
   GP2:
	UF : 1, UT : 1,
	J1=    90.000 deg,	J2=     -.000 deg
};
P[42]{
   GP1:
	UF : 1, UT : 1,		CONFIG : 'N U T, 0, 0, 0',
	X =  2771.051  mm,	Y =    52.392  mm,	Z =  -583.085  mm,
	W =   -14.706 deg,	P =    41.251 deg,	R =    68.262 deg
   GP2:
	UF : 1, UT : 1,
	J1=    90.000 deg,	J2=     -.000 deg
};
P[43]{
   GP1:
	UF : 1, UT : 1,		CONFIG : 'N U T, 0, 0, 0',
	X =  2773.300  mm,	Y =   -46.177  mm,	Z =  -424.688  mm,
	W =    -3.866 deg,	P =    15.387 deg,	R =   -14.287 deg
   GP2:
	UF : 1, UT : 1,
	J1=    90.000 deg,	J2=     0.000 deg
};
P[44]{
   GP1:
	UF : 1, UT : 1,		CONFIG : 'N U T, 0, 0, 0',
	X =  2388.156  mm,	Y =   -46.177  mm,	Z =   494.312  mm,
	W =    -3.866 deg,	P =    15.387 deg,	R =   -14.287 deg
   GP2:
	UF : 1, UT : 1,
	J1=    90.000 deg,	J2=     0.000 deg
};
P[45]{
   GP1:
	UF : 1, UT : 1,		CONFIG : 'N U T, 0, 0, 0',
	X =  2665.300  mm,	Y =   191.823  mm,	Z =   494.312  mm,
	W =    34.617 deg,	P =    32.086 deg,	R =   -37.579 deg
   GP2:
	UF : 1, UT : 1,
	J1=    90.000 deg,	J2=     0.000 deg
};
P[46]{
   GP1:
	UF : 1, UT : 1,		CONFIG : 'N U T, 0, 0, 0',
	X =  2746.301  mm,	Y =   359.823  mm,	Z =   372.313  mm,
	W =    44.065 deg,	P =    13.982 deg,	R =   -14.016 deg
   GP2:
	UF : 1, UT : 1,
	J1=    90.000 deg,	J2=     0.000 deg
};
P[47]{
   GP1:
	UF : 1, UT : 1,		CONFIG : 'N U T, 0, 0, 0',
	X =  2775.572  mm,	Y =    45.614  mm,	Z =  -584.321  mm,
	W =    -7.893 deg,	P =    29.549 deg,	R =   -15.873 deg
   GP2:
	UF : 1, UT : 1,
	J1=    90.000 deg,	J2=     -.000 deg
};
P[48]{
   GP1:
	UF : 1, UT : 1,		CONFIG : 'N U T, 0, 0, 0',
	X =  2775.432  mm,	Y =   -50.618  mm,	Z =  -585.269  mm,
	W =    -7.969 deg,	P =    29.524 deg,	R =   -15.865 deg
   GP2:
	UF : 1, UT : 1,
	J1=    90.000 deg,	J2=     -.000 deg
};
P[49]{
   GP1:
	UF : 1, UT : 1,		CONFIG : 'N U T, 0, 0, 0',
	X =  2711.142  mm,	Y =   208.547  mm,	Z =   521.702  mm,
	W =    43.274 deg,	P =    13.788 deg,	R =   -14.206 deg
   GP2:
	UF : 1, UT : 1,
	J1=    90.000 deg,	J2=     0.000 deg
};
P[50]{
   GP1:
	UF : 1, UT : 1,		CONFIG : 'N U T, 0, 0, 0',
	X =  2711.142  mm,	Y =  -358.128  mm,	Z =   441.702  mm,
	W =   -43.273 deg,	P =   -13.788 deg,	R =   -14.206 deg
   GP2:
	UF : 1, UT : 1,
	J1=    90.000 deg,	J2=     0.000 deg
};
P[51]{
   GP1:
	UF : 1, UT : 1,		CONFIG : 'N U T, 0, 0, 0',
	X =  2754.975  mm,	Y =   412.754  mm,	Z =   328.449  mm,
	W =    43.280 deg,	P =    13.791 deg,	R =   -11.854 deg
   GP2:
	UF : 1, UT : 1,
	J1=    90.000 deg,	J2=     0.000 deg
};
P[52]{
   GP1:
	UF : 1, UT : 1,		CONFIG : 'N U T, 0, 0, 0',
	X =  2709.583  mm,	Y =   412.578  mm,	Z =   327.552  mm,
	W =    43.277 deg,	P =    13.792 deg,	R =   -10.715 deg
   GP2:
	UF : 1, UT : 1,
	J1=    90.000 deg,	J2=     0.000 deg
};
P[53]{
   GP1:
	UF : 1, UT : 1,		CONFIG : 'N U T, 0, 0, 0',
	X =  2711.772  mm,	Y =  -257.488  mm,	Z =   482.569  mm,
	W =   -43.274 deg,	P =   -13.788 deg,	R =   -14.206 deg
   GP2:
	UF : 1, UT : 1,
	J1=    90.000 deg,	J2=     0.000 deg
};
P[54]{
   GP1:
	UF : 1, UT : 1,		CONFIG : 'F U T, 0, 0, 0',
	X =  2682.821  mm,	Y =   109.226  mm,	Z =   556.209  mm,
	W =     6.709 deg,	P =   -51.514 deg,	R =    -2.307 deg
   GP2:
	UF : 1, UT : 1,
	J1=    90.000 deg,	J2=     0.000 deg
};
P[55]{
   GP1:
	UF : 1, UT : 1,		CONFIG : 'F U T, 0, 0, 0',
	X =  2878.931  mm,	Y =   284.681  mm,	Z =   359.593  mm,
	W =    -2.366 deg,	P =   -44.781 deg,	R =    15.348 deg
   GP2:
	UF : 1, UT : 1,
	J1=    90.000 deg,	J2=     0.000 deg
};
P[56]{
   GP1:
	UF : 1, UT : 1,		CONFIG : 'N U T, 0, 0, 0',
	X =  2755.648  mm,	Y =  -419.671  mm,	Z =   324.655  mm,
	W =   -43.273 deg,	P =   -13.781 deg,	R =   -15.654 deg
   GP2:
	UF : 1, UT : 1,
	J1=    90.000 deg,	J2=     0.000 deg
};
P[57]{
   GP1:
	UF : 1, UT : 1,		CONFIG : 'N U T, 0, 0, 0',
	X =  2707.716  mm,	Y =  -419.404  mm,	Z =   324.423  mm,
	W =   -43.229 deg,	P =   -13.780 deg,	R =   -15.681 deg
   GP2:
	UF : 1, UT : 1,
	J1=    90.000 deg,	J2=     0.000 deg
};
P[58]{
   GP1:
	UF : 1, UT : 1,		CONFIG : 'F U T, 0, 0, 0',
	X =  2900.602  mm,	Y =   280.855  mm,	Z =   330.798  mm,
	W =    -2.362 deg,	P =   -44.780 deg,	R =    15.343 deg
   GP2:
	UF : 1, UT : 1,
	J1=    90.000 deg,	J2=     0.000 deg
};
P[59]{
   GP1:
	UF : 1, UT : 1,		CONFIG : 'F U T, 0, 0, 0',
	X =  2688.926  mm,	Y =   145.792  mm,	Z =   479.238  mm,
	W =    11.537 deg,	P =   -44.440 deg,	R =    16.356 deg
   GP2:
	UF : 1, UT : 1,
	J1=    90.000 deg,	J2=     0.000 deg
};
P[60]{
   GP1:
	UF : 1, UT : 1,		CONFIG : 'F U T, 0, 0, 0',
	X =  2901.607  mm,	Y =   353.529  mm,	Z =   330.605  mm,
	W =    -2.363 deg,	P =   -44.778 deg,	R =    21.461 deg
   GP2:
	UF : 1, UT : 1,
	J1=    90.000 deg,	J2=     0.000 deg
};
P[61]{
   GP1:
	UF : 1, UT : 1,		CONFIG : 'F U T, 0, 0, 0',
	X =  2822.856  mm,	Y =   307.220  mm,	Z =   422.096  mm,
	W =    11.538 deg,	P =   -44.441 deg,	R =    36.427 deg
   GP2:
	UF : 1, UT : 1,
	J1=    90.000 deg,	J2=     0.000 deg
};
P[62]{
   GP1:
	UF : 1, UT : 1,		CONFIG : 'F U T, 0, 0, 0',
	X =  2901.149  mm,	Y =   394.270  mm,	Z =   330.773  mm,
	W =     3.865 deg,	P =   -44.777 deg,	R =    31.534 deg
   GP2:
	UF : 1, UT : 1,
	J1=    90.000 deg,	J2=     0.000 deg
};
P[63]{
   GP1:
	UF : 1, UT : 1,		CONFIG : 'N U T, 0, 0, 0',
	X =  2506.771  mm,	Y =    -3.468  mm,	Z =   625.975  mm,
	W =   -10.413 deg,	P =   -54.310 deg,	R =     6.585 deg
   GP2:
	UF : 1, UT : 1,
	J1=    90.000 deg,	J2=     0.000 deg
};
P[64]{
   GP1:
	UF : 1, UT : 1,		CONFIG : 'N U T, 0, 0, 0',
	X =  2876.416  mm,	Y =  -294.248  mm,	Z =   360.831  mm,
	W =    12.831 deg,	P =   -43.281 deg,	R =   -27.682 deg
   GP2:
	UF : 1, UT : 1,
	J1=    90.000 deg,	J2=     0.000 deg
};
P[65]{
   GP1:
	UF : 1, UT : 1,		CONFIG : 'F U T, 0, 0, 0',
	X =  2896.882  mm,	Y =   404.532  mm,	Z =   330.811  mm,
	W =     3.880 deg,	P =   -44.778 deg,	R =    44.019 deg
   GP2:
	UF : 1, UT : 1,
	J1=    89.999 deg,	J2=     0.000 deg
};
P[66]{
   GP1:
	UF : 1, UT : 1,		CONFIG : 'F U T, 0, 0, 0',
	X =  2875.458  mm,	Y =   411.451  mm,	Z =   330.775  mm,
	W =    11.523 deg,	P =   -44.430 deg,	R =    62.752 deg
   GP2:
	UF : 1, UT : 1,
	J1=    89.999 deg,	J2=     0.000 deg
};
P[67]{
   GP1:
	UF : 1, UT : 1,		CONFIG : 'N U T, 0, 0, 0',
	X =  2901.594  mm,	Y =  -286.321  mm,	Z =   331.051  mm,
	W =    12.831 deg,	P =   -43.281 deg,	R =   -27.681 deg
   GP2:
	UF : 1, UT : 1,
	J1=    90.000 deg,	J2=     0.000 deg
};
P[68]{
   GP1:
	UF : 1, UT : 1,		CONFIG : 'N U T, 0, 0, 0',
	X =  2657.003  mm,	Y =   -63.546  mm,	Z =   568.894  mm,
	W =     -.758 deg,	P =   -43.272 deg,	R =    -9.466 deg
   GP2:
	UF : 1, UT : 1,
	J1=    90.000 deg,	J2=     0.000 deg
};
P[69]{
   GP1:
	UF : 1, UT : 1,		CONFIG : 'N U T, 0, 0, 0',
	X =  2901.299  mm,	Y =  -359.339  mm,	Z =   331.905  mm,
	W =    12.831 deg,	P =   -43.281 deg,	R =   -27.681 deg
   GP2:
	UF : 1, UT : 1,
	J1=    90.000 deg,	J2=     0.000 deg
};
P[70]{
   GP1:
	UF : 1, UT : 1,		CONFIG : 'N U T, 0, 0, 0',
	X =  2795.455  mm,	Y =  -317.713  mm,	Z =   407.823  mm,
	W =     -.758 deg,	P =   -43.273 deg,	R =   -36.153 deg
   GP2:
	UF : 1, UT : 1,
	J1=    90.000 deg,	J2=     0.000 deg
};
P[71]{
   GP1:
	UF : 1, UT : 1,		CONFIG : 'F U T, 0, 0, 0',
	X =  2626.454  mm,	Y =    58.795  mm,	Z =   612.721  mm,
	W =    10.455 deg,	P =   -53.174 deg,	R =    -8.186 deg
   GP2:
	UF : 1, UT : 1,
	J1=    90.000 deg,	J2=     0.000 deg
};
P[72]{
   GP1:
	UF : 1, UT : 1,		CONFIG : 'N U T, 0, 0, 0',
	X =  2902.274  mm,	Y =  -399.677  mm,	Z =   330.687  mm,
	W =     3.818 deg,	P =   -42.738 deg,	R =   -27.631 deg
   GP2:
	UF : 1, UT : 1,
	J1=    90.000 deg,	J2=     0.000 deg
};
P[73]{
   GP1:
	UF : 1, UT : 1,		CONFIG : 'N U T, 0, 0, 0',
	X =  2112.950  mm,	Y =   371.014  mm,	Z =  1254.690  mm,
	W =     3.998 deg,	P =    -8.968 deg,	R =   -24.204 deg
   GP2:
	UF : 1, UT : 1,
	J1=   135.000 deg,	J2=     0.000 deg
};
P[74]{
   GP1:
	UF : 1, UT : 1,		CONFIG : 'F U T, 0, 0, 0',
	X =  2878.931  mm,	Y =   284.681  mm,	Z =   359.593  mm,
	W =    -2.366 deg,	P =   -44.781 deg,	R =    15.348 deg
   GP2:
	UF : 1, UT : 1,
	J1=    90.000 deg,	J2=     0.000 deg
};
P[75]{
   GP1:
	UF : 1, UT : 1,		CONFIG : 'N U T, 0, 0, 0',
	X =  2894.061  mm,	Y =  -412.034  mm,	Z =   330.685  mm,
	W =    -2.363 deg,	P =   -42.893 deg,	R =   -45.036 deg
   GP2:
	UF : 1, UT : 1,
	J1=    90.000 deg,	J2=     0.000 deg
};
P[76]{
   GP1:
	UF : 1, UT : 1,		CONFIG : 'N U T, 0, 0, 0',
	X =  2348.894  mm,	Y =   386.121  mm,	Z =   308.013  mm,
	W =    44.432 deg,	P =     8.082 deg,	R =   -31.054 deg
   GP2:
	UF : 1, UT : 1,
	J1=     0.000 deg,	J2=   180.000 deg
};
P[77]{
   GP1:
	UF : 1, UT : 1,		CONFIG : 'N U T, 0, 0, 0',
	X =  2878.275  mm,	Y =  -416.748  mm,	Z =   330.172  mm,
	W =     -.758 deg,	P =   -43.274 deg,	R =   -72.516 deg
   GP2:
	UF : 1, UT : 1,
	J1=    90.000 deg,	J2=     0.000 deg
};
P[78]{
   GP1:
	UF : 1, UT : 1,		CONFIG : 'N U T, 0, 0, 0',
	X =  2111.886  mm,	Y =     7.673  mm,	Z =  1193.435  mm,
	W =    -1.732 deg,	P =    -2.297 deg,	R =   -23.799 deg
   GP2:
	UF : 1, UT : 1,
	J1=   135.000 deg,	J2=     0.000 deg
};
P[79]{
   GP1:
	UF : 1, UT : 1,		CONFIG : 'N U T, 0, 0, 0',
	X =  2111.696  mm,	Y =  -402.392  mm,	Z =  1193.417  mm,
	W =    -1.735 deg,	P =    -2.297 deg,	R =   -23.794 deg
   GP2:
	UF : 1, UT : 1,
	J1=   135.000 deg,	J2=     0.000 deg
};
P[80]{
   GP1:
	UF : 1, UT : 1,		CONFIG : 'F U T, 0, 0, 0',
	X =  2822.856  mm,	Y =   307.220  mm,	Z =   422.096  mm,
	W =    11.538 deg,	P =   -44.441 deg,	R =    36.427 deg
   GP2:
	UF : 1, UT : 1,
	J1=    90.000 deg,	J2=     0.000 deg
};
P[81]{
   GP1:
	UF : 1, UT : 1,		CONFIG : 'F U T, 0, 0, 0',
	X =  2626.454  mm,	Y =    58.795  mm,	Z =   612.721  mm,
	W =    10.455 deg,	P =   -53.174 deg,	R =    -8.186 deg
   GP2:
	UF : 1, UT : 1,
	J1=    90.000 deg,	J2=     0.000 deg
};
P[82]{
   GP1:
	UF : 1, UT : 1,		CONFIG : 'F U T, 0, 0, 0',
	X =  2878.931  mm,	Y =   284.681  mm,	Z =   359.593  mm,
	W =    -2.366 deg,	P =   -44.781 deg,	R =    15.348 deg
   GP2:
	UF : 1, UT : 1,
	J1=    90.000 deg,	J2=     0.000 deg
};
P[83]{
   GP1:
	UF : 1, UT : 1,		CONFIG : 'F U T, 0, 0, 0',
	X =  2822.856  mm,	Y =   307.220  mm,	Z =   422.096  mm,
	W =    11.538 deg,	P =   -44.441 deg,	R =    36.427 deg
   GP2:
	UF : 1, UT : 1,
	J1=    90.000 deg,	J2=     0.000 deg
};
P[84]{
   GP1:
	UF : 1, UT : 1,		CONFIG : 'F U T, 0, 0, 0',
	X =  2688.926  mm,	Y =   145.792  mm,	Z =   479.238  mm,
	W =    11.537 deg,	P =   -44.440 deg,	R =    16.356 deg
   GP2:
	UF : 1, UT : 1,
	J1=    90.000 deg,	J2=     0.000 deg
};
P[85]{
   GP1:
	UF : 1, UT : 1,		CONFIG : 'N U T, 0, 0, 0',
	X =  2506.771  mm,	Y =    -3.468  mm,	Z =   625.975  mm,
	W =   -10.413 deg,	P =   -54.310 deg,	R =     6.585 deg
   GP2:
	UF : 1, UT : 1,
	J1=    90.000 deg,	J2=     0.000 deg
};
P[86]{
   GP1:
	UF : 1, UT : 1,		CONFIG : 'N U T, 0, 0, 0',
	X =  2876.416  mm,	Y =  -294.248  mm,	Z =   360.831  mm,
	W =    12.831 deg,	P =   -43.281 deg,	R =   -27.682 deg
   GP2:
	UF : 1, UT : 1,
	J1=    90.000 deg,	J2=     0.000 deg
};
P[87]{
   GP1:
	UF : 1, UT : 1,		CONFIG : 'N U T, 0, 0, 0',
	X =  2795.455  mm,	Y =  -317.713  mm,	Z =   407.823  mm,
	W =     -.758 deg,	P =   -43.273 deg,	R =   -36.153 deg
   GP2:
	UF : 1, UT : 1,
	J1=    90.000 deg,	J2=     0.000 deg
};
P[88]{
   GP1:
	UF : 1, UT : 1,		CONFIG : 'N U T, 0, 0, 0',
	X =  2774.022  mm,	Y =  -241.428  mm,	Z =   477.421  mm,
	W =      .369 deg,	P =   -45.174 deg,	R =   -28.340 deg
   GP2:
	UF : 1, UT : 1,
	J1=    90.000 deg,	J2=     0.000 deg
};
P[89]{
   GP1:
	UF : 1, UT : 1,		CONFIG : 'N U T, 0, 0, 0',
	X =  2876.416  mm,	Y =  -294.248  mm,	Z =   360.831  mm,
	W =    12.831 deg,	P =   -43.281 deg,	R =   -27.682 deg
   GP2:
	UF : 1, UT : 1,
	J1=    90.000 deg,	J2=     0.000 deg
};
P[90]{
   GP1:
	UF : 1, UT : 1,		CONFIG : 'N U T, 0, 0, 0',
	X =  2795.455  mm,	Y =  -317.713  mm,	Z =   431.916  mm,
	W =    16.615 deg,	P =   -40.558 deg,	R =   -61.910 deg
   GP2:
	UF : 1, UT : 1,
	J1=    90.000 deg,	J2=     0.000 deg
};
P[91]{
   GP1:
	UF : 1, UT : 1,		CONFIG : 'N U T, 0, 0, 0',
	X =  1233.935  mm,	Y = -1549.119  mm,	Z =  1652.621  mm,
	W =   -59.729 deg,	P =   -13.841 deg,	R =    34.854 deg
   GP2:
	UF : 1, UT : 1,
	J1=   180.000 deg,	J2=  -125.000 deg
};
P[92]{
   GP1:
	UF : 1, UT : 1,		CONFIG : 'N U T, 0, 0, -1',
	X =  2284.571  mm,	Y =   224.723  mm,	Z =  -103.907  mm,
	W =    -1.824 deg,	P =    43.273 deg,	R =  -177.941 deg
   GP2:
	UF : 1, UT : 1,
	J1=     0.000 deg,	J2=   180.000 deg
};
P[93]{
   GP1:
	UF : 1, UT : 1,		CONFIG : 'N U T, 0, 0, 0',
	X =  2865.354  mm,	Y =  1371.120  mm,	Z =    50.536  mm,
	W =    -1.528 deg,	P =    -1.642 deg,	R =     2.928 deg
   GP2:
	UF : 1, UT : 1,
	J1=    94.999 deg,	J2=    90.000 deg
};
P[94]{
   GP1:
	UF : 1, UT : 1,		CONFIG : 'N U T, 0, 0, 0',
	X =  1724.172  mm,	Y =   -99.215  mm,	Z =   441.840  mm,
	W =    -3.538 deg,	P =   -37.455 deg,	R =   -26.472 deg
   GP2:
	UF : 1, UT : 1,
	J1=     0.000 deg,	J2=   180.000 deg
};
P[95]{
   GP1:
	UF : 1, UT : 1,		CONFIG : 'N U T, 0, 0, 0',
	X =  2094.232  mm,	Y =    19.822  mm,	Z =    16.623  mm,
	W =   -33.555 deg,	P =   -20.475 deg,	R =   113.896 deg
   GP2:
	UF : 1, UT : 1,
	J1=    80.000 deg,	J2=    90.000 deg
};
P[96]{
   GP1:
	UF : 1, UT : 1,		CONFIG : 'N U T, 0, 0, 0',
	X =  2865.354  mm,	Y =  1351.052  mm,	Z =    50.536  mm,
	W =    -1.528 deg,	P =    -1.642 deg,	R =     2.928 deg
   GP2:
	UF : 1, UT : 1,
	J1=    94.999 deg,	J2=    90.000 deg
};
P[97]{
   GP1:
	UF : 1, UT : 1,		CONFIG : 'N U T, 0, 0, 0',
	X =  2206.375  mm,	Y =   -84.206  mm,	Z =    -4.653  mm,
	W =   -33.592 deg,	P =   -20.528 deg,	R =   117.916 deg
   GP2:
	UF : 1, UT : 1,
	J1=    80.000 deg,	J2=    90.000 deg
};
P[98]{
   GP1:
	UF : 1, UT : 1,		CONFIG : 'N U T, 0, 0, 0',
	X =  2849.008  mm,	Y =  1361.478  mm,	Z =    50.536  mm,
	W =    -1.528 deg,	P =    -1.642 deg,	R =     2.928 deg
   GP2:
	UF : 1, UT : 1,
	J1=    94.999 deg,	J2=    90.000 deg
};
P[99]{
   GP1:
	UF : 1, UT : 1,		CONFIG : 'N U T, 0, 0, 0',
	X =  2031.518  mm,	Y =    20.497  mm,	Z =     8.683  mm,
	W =    38.911 deg,	P =    24.670 deg,	R =    12.953 deg
   GP2:
	UF : 1, UT : 1,
	J1=    90.000 deg,	J2=    90.000 deg
};
P[100]{
   GP1:
	UF : 1, UT : 1,		CONFIG : 'N U T, 0, 0, 0',
	X =  2255.454  mm,	Y =  -121.848  mm,	Z =   -10.027  mm,
	W =   -17.164 deg,	P =   -39.269 deg,	R =    90.811 deg
   GP2:
	UF : 1, UT : 1,
	J1=    80.000 deg,	J2=    90.000 deg
};
P[101]{
   GP1:
	UF : 1, UT : 1,		CONFIG : 'N U T, 0, 0, 0',
	X =  2303.774  mm,	Y =  -139.202  mm,	Z =   -19.217  mm,
	W =   -17.185 deg,	P =   -39.290 deg,	R =    99.791 deg
   GP2:
	UF : 1, UT : 1,
	J1=    80.000 deg,	J2=    90.000 deg
};
P[102]{
   GP1:
	UF : 1, UT : 1,		CONFIG : 'N U T, 0, 0, 0',
	X =  2624.706  mm,	Y =  -150.826  mm,	Z =   504.595  mm,
	W =    29.842 deg,	P =    35.744 deg,	R =  -141.857 deg
   GP2:
	UF : 1, UT : 1,
	J1=    90.000 deg,	J2=     0.000 deg
};
P[103]{
   GP1:
	UF : 1, UT : 1,		CONFIG : 'N U T, 0, 0, 0',
	X =  2683.383  mm,	Y =  -300.218  mm,	Z =   394.001  mm,
	W =    31.985 deg,	P =    33.748 deg,	R =  -135.954 deg
   GP2:
	UF : 1, UT : 1,
	J1=    90.000 deg,	J2=     0.000 deg
};
P[104]{
   GP1:
	UF : 1, UT : 1,		CONFIG : 'N U T, 0, 0, 0',
	X =  2319.749  mm,	Y =  -144.824  mm,	Z =   -20.315  mm,
	W =   -25.651 deg,	P =   -34.890 deg,	R =    98.088 deg
   GP2:
	UF : 1, UT : 1,
	J1=    80.000 deg,	J2=    90.000 deg
};
P[105]{
   GP1:
	UF : 1, UT : 1,		CONFIG : 'N U T, 0, 0, 0',
	X =  2336.580  mm,	Y =  -147.632  mm,	Z =   -22.463  mm,
	W =   -25.652 deg,	P =   -34.890 deg,	R =    87.210 deg
   GP2:
	UF : 1, UT : 1,
	J1=    80.000 deg,	J2=    90.000 deg
};
P[106]{
   GP1:
	UF : 1, UT : 1,		CONFIG : 'N U T, 0, 0, 0',
	X =  2333.007  mm,	Y =  -148.653  mm,	Z =   -24.467  mm,
	W =    -6.859 deg,	P =   -41.860 deg,	R =   116.724 deg
   GP2:
	UF : 1, UT : 1,
	J1=    80.000 deg,	J2=    90.000 deg
};
P[107]{
   GP1:
	UF : 1, UT : 1,		CONFIG : 'N U T, 0, 0, 0',
	X =  2355.906  mm,	Y =  -150.954  mm,	Z =   -27.328  mm,
	W =   -13.723 deg,	P =   -38.566 deg,	R =   105.555 deg
   GP2:
	UF : 1, UT : 1,
	J1=    80.000 deg,	J2=    90.000 deg
};
P[108]{
   GP1:
	UF : 1, UT : 1,		CONFIG : 'N U T, 0, 0, 0',
	X =  2780.517  mm,	Y =  -372.561  mm,	Z =   464.471  mm,
	W =    32.643 deg,	P =     1.822 deg,	R =   -93.819 deg
   GP2:
	UF : 1, UT : 1,
	J1=    90.000 deg,	J2=     0.000 deg
};
P[109]{
   GP1:
	UF : 1, UT : 1,		CONFIG : 'N U T, 0, 0, 0',
	X =  2543.169  mm,	Y =  -170.233  mm,	Z =   459.679  mm,
	W =    15.320 deg,	P =    20.551 deg,	R =  -109.367 deg
   GP2:
	UF : 1, UT : 1,
	J1=    90.000 deg,	J2=     0.000 deg
};
P[110]{
   GP1:
	UF : 1, UT : 1,		CONFIG : 'N U T, 0, 0, 0',
	X =  2564.790  mm,	Y =   179.821  mm,	Z =   472.963  mm,
	W =   -33.661 deg,	P =    20.429 deg,	R =   124.430 deg
   GP2:
	UF : 1, UT : 1,
	J1=    90.000 deg,	J2=     0.000 deg
};
P[111]{
   GP1:
	UF : 1, UT : 1,		CONFIG : 'N U T, 0, 0, 0',
	X =  2655.463  mm,	Y =   284.548  mm,	Z =   472.963  mm,
	W =   -37.578 deg,	P =    10.941 deg,	R =   104.868 deg
   GP2:
	UF : 1, UT : 1,
	J1=    90.000 deg,	J2=     0.000 deg
};
P[112]{
   GP1:
	UF : 1, UT : 1,		CONFIG : 'N U T, 0, 0, 0',
	X =  2588.366  mm,	Y =  -191.938  mm,	Z =   -64.016  mm,
	W =    39.677 deg,	P =   -13.111 deg,	R =    10.485 deg
   GP2:
	UF : 1, UT : 1,
	J1=    80.000 deg,	J2=    90.000 deg
};
P[113]{
   GP1:
	UF : 1, UT : 1,		CONFIG : 'N U T, 0, 0, 0',
	X =  2634.096  mm,	Y =  -220.389  mm,	Z =   -70.040  mm,
	W =    17.668 deg,	P =   -27.967 deg,	R =      .790 deg
   GP2:
	UF : 1, UT : 1,
	J1=    80.000 deg,	J2=    90.000 deg
};
P[114]{
   GP1:
	UF : 1, UT : 1,		CONFIG : 'N U T, 0, 0, 0',
	X =  2635.327  mm,	Y =  -279.131  mm,	Z =   -74.721  mm,
	W =   -36.832 deg,	P =     1.847 deg,	R =    73.287 deg
   GP2:
	UF : 1, UT : 1,
	J1=    80.000 deg,	J2=    90.000 deg
};
P[115]{
   GP1:
	UF : 1, UT : 1,		CONFIG : 'N U T, 0, 0, 0',
	X =  2628.236  mm,	Y =  -300.399  mm,	Z =   -74.071  mm,
	W =   -38.135 deg,	P =     7.631 deg,	R =    72.017 deg
   GP2:
	UF : 1, UT : 1,
	J1=    80.000 deg,	J2=    90.000 deg
};
P[116]{
   GP1:
	UF : 1, UT : 1,		CONFIG : 'N U T, 0, 0, 0',
	X =  2727.478  mm,	Y =   349.696  mm,	Z =   477.126  mm,
	W =   -21.853 deg,	P =    13.056 deg,	R =    95.740 deg
   GP2:
	UF : 1, UT : 1,
	J1=    90.000 deg,	J2=     0.000 deg
};
P[117]{
   GP1:
	UF : 1, UT : 1,		CONFIG : 'N U T, 0, 0, 0',
	X =  1988.908  mm,	Y =   131.267  mm,	Z =   609.126  mm,
	W =    17.833 deg,	P =    51.565 deg,	R =    17.002 deg
   GP2:
	UF : 1, UT : 1,
	J1=    90.000 deg,	J2=     0.000 deg
};
P[118]{
   GP1:
	UF : 1, UT : 1,		CONFIG : 'N U T, 0, 0, 0',
	X =  1707.576  mm,	Y =   131.267  mm,	Z =   438.126  mm,
	W =    17.833 deg,	P =    51.565 deg,	R =    17.002 deg
   GP2:
	UF : 1, UT : 1,
	J1=    90.000 deg,	J2=     0.000 deg
};
P[119]{
   GP1:
	UF : 1, UT : 1,		CONFIG : 'N U T, 0, 0, 0',
	X =  2625.099  mm,	Y =  -317.058  mm,	Z =   -72.888  mm,
	W =   -38.026 deg,	P =     5.892 deg,	R =    87.515 deg
   GP2:
	UF : 1, UT : 1,
	J1=    80.000 deg,	J2=    90.000 deg
};
P[120]{
   GP1:
	UF : 1, UT : 1,		CONFIG : 'N U T, 0, 0, 0',
	X =  2625.646  mm,	Y =  -569.480  mm,	Z =   -73.369  mm,
	W =   -38.231 deg,	P =   -10.585 deg,	R =    66.882 deg
   GP2:
	UF : 1, UT : 1,
	J1=    80.000 deg,	J2=    90.000 deg
};
P[121]{
   GP1:
	UF : 1, UT : 1,		CONFIG : 'N U T, 0, 0, 0',
	X =  1813.192  mm,	Y =   169.381  mm,	Z =   514.495  mm,
	W =    10.023 deg,	P =    44.106 deg,	R =    14.249 deg
   GP2:
	UF : 1, UT : 1,
	J1=    90.000 deg,	J2=     0.000 deg
};
P[122]{
   GP1:
	UF : 1, UT : 1,		CONFIG : 'N U T, 0, 0, 0',
	X =  1731.370  mm,	Y =  -138.313  mm,	Z =   432.673  mm,
	W =   -27.009 deg,	P =    37.471 deg,	R =   -39.958 deg
   GP2:
	UF : 1, UT : 1,
	J1=    90.000 deg,	J2=     0.000 deg
};
P[123]{
   GP1:
	UF : 1, UT : 1,		CONFIG : 'N U T, 0, 0, 0',
	X =  2381.736  mm,	Y =  -370.018  mm,	Z =   191.729  mm,
	W =    -3.680 deg,	P =     -.881 deg,	R =   -13.566 deg
   GP2:
	UF : 1, UT : 1,
	J1=    90.000 deg,	J2=  -135.000 deg
};
P[124]{
   GP1:
	UF : 1, UT : 1,		CONFIG : 'N U T, 0, 0, 1',
	X =  2741.800  mm,	Y =  -291.447  mm,	Z =   327.230  mm,
	W =    29.206 deg,	P =    34.602 deg,	R =  -135.393 deg
   GP2:
	UF : 1, UT : 1,
	J1=    90.000 deg,	J2=     0.000 deg
};
P[125]{
   GP1:
	UF : 1, UT : 1,		CONFIG : 'N U T, 0, 0, 0',
	X =  1763.068  mm,	Y =  -201.487  mm,	Z =   455.614  mm,
	W =   -27.009 deg,	P =    37.471 deg,	R =   -39.958 deg
   GP2:
	UF : 1, UT : 1,
	J1=    90.000 deg,	J2=     0.000 deg
};
P[126]{
   GP1:
	UF : 1, UT : 1,		CONFIG : 'N U T, 0, 0, 0',
	X =  1763.068  mm,	Y =    25.303  mm,	Z =   455.614  mm,
	W =     5.616 deg,	P =    44.724 deg,	R =     7.956 deg
   GP2:
	UF : 1, UT : 1,
	J1=    90.000 deg,	J2=     0.000 deg
};
P[127]{
   GP1:
	UF : 1, UT : 1,		CONFIG : 'N U T, 0, 0, 0',
	X =  1813.067  mm,	Y =  -148.698  mm,	Z =   975.615  mm,
	W =     0.000 deg,	P =      .001 deg,	R =     5.643 deg
   GP2:
	UF : 1, UT : 1,
	J1=    45.000 deg,	J2=     0.000 deg
};
P[128]{
   GP1:
	UF : 1, UT : 1,		CONFIG : 'N U T, 0, 0, 1',
	X =  2742.971  mm,	Y =  -340.891  mm,	Z =   327.062  mm,
	W =    30.065 deg,	P =    35.210 deg,	R =  -134.887 deg
   GP2:
	UF : 1, UT : 1,
	J1=    90.000 deg,	J2=     0.000 deg
};
P[129]{
   GP1:
	UF : 1, UT : 1,		CONFIG : 'N U T, 0, 0, 1',
	X =  2759.544  mm,	Y =  -364.993  mm,	Z =   329.461  mm,
	W =    28.607 deg,	P =    30.691 deg,	R =  -111.066 deg
   GP2:
	UF : 1, UT : 1,
	J1=    90.000 deg,	J2=     0.000 deg
};
P[130]{
   GP1:
	UF : 1, UT : 1,		CONFIG : 'N U T, 0, 0, 0',
	X =  1813.067  mm,	Y =  -143.179  mm,	Z =  1084.186  mm,
	W =     0.000 deg,	P =      .001 deg,	R =     5.643 deg
   GP2:
	UF : 1, UT : 1,
	J1=    45.000 deg,	J2=     0.000 deg
};
P[131]{
   GP1:
	UF : 1, UT : 1,		CONFIG : 'N U T, 0, 0, 0',
	X =  1813.067  mm,	Y =   375.821  mm,	Z =   983.186  mm,
	W =     0.000 deg,	P =      .001 deg,	R =     5.643 deg
   GP2:
	UF : 1, UT : 1,
	J1=    45.000 deg,	J2=     0.000 deg
};
P[132]{
   GP1:
	UF : 1, UT : 1,		CONFIG : 'N U T, 0, 0, 1',
	X =  2774.975  mm,	Y =  -367.824  mm,	Z =   328.645  mm,
	W =    30.303 deg,	P =    27.056 deg,	R =   -98.836 deg
   GP2:
	UF : 1, UT : 1,
	J1=    90.000 deg,	J2=     0.000 deg
};
P[133]{
   GP1:
	UF : 1, UT : 1,		CONFIG : 'N U T, 0, 0, 0',
	X =  2741.560  mm,	Y =   284.208  mm,	Z =   324.647  mm,
	W =   -43.506 deg,	P =    12.857 deg,	R =   103.193 deg
   GP2:
	UF : 1, UT : 1,
	J1=    90.000 deg,	J2=     0.000 deg
};
P[134]{
   GP1:
	UF : 1, UT : 1,		CONFIG : 'N U T, 0, 0, 0',
	X =  1817.884  mm,	Y =   125.453  mm,	Z =  1218.185  mm,
	W =     0.000 deg,	P =      .001 deg,	R =     5.643 deg
   GP2:
	UF : 1, UT : 1,
	J1=    45.000 deg,	J2=     0.000 deg
};
P[135]{
   GP1:
	UF : 1, UT : 1,		CONFIG : 'N U T, 0, 0, 0',
	X =   922.650  mm,	Y =   428.778  mm,	Z =  1743.265  mm,
	W =    20.739 deg,	P =   -18.803 deg,	R =   -28.768 deg
   GP2:
	UF : 1, UT : 1,
	J1=   135.000 deg,	J2=     0.000 deg
};
P[136]{
   GP1:
	UF : 1, UT : 1,		CONFIG : 'N U T, 0, 0, 0',
	X =  1379.547  mm,	Y =   574.325  mm,	Z =  1305.023  mm,
	W =     8.340 deg,	P =   -18.155 deg,	R =   -25.224 deg
   GP2:
	UF : 1, UT : 1,
	J1=   135.000 deg,	J2=     0.000 deg
};
P[137]{
   GP1:
	UF : 1, UT : 1,		CONFIG : 'N U T, 0, 0, 0',
	X =  2100.617  mm,	Y =   614.231  mm,	Z =  1305.022  mm,
	W =    13.075 deg,	P =   -27.074 deg,	R =   -27.053 deg
   GP2:
	UF : 1, UT : 1,
	J1=   135.000 deg,	J2=     0.000 deg
};
P[138]{
   GP1:
	UF : 1, UT : 1,		CONFIG : 'N U T, 0, 0, 0',
	X =  2741.909  mm,	Y =   330.818  mm,	Z =   325.255  mm,
	W =   -43.506 deg,	P =    12.857 deg,	R =   103.193 deg
   GP2:
	UF : 1, UT : 1,
	J1=    90.000 deg,	J2=     0.000 deg
};
P[139]{
   GP1:
	UF : 1, UT : 1,		CONFIG : 'N U T, 0, 0, 0',
	X =  2752.167  mm,	Y =   352.560  mm,	Z =   324.676  mm,
	W =   -20.735 deg,	P =    23.320 deg,	R =    96.090 deg
   GP2:
	UF : 1, UT : 1,
	J1=    90.000 deg,	J2=     0.000 deg
};
P[140]{
   GP1:
	UF : 1, UT : 1,		CONFIG : 'N U T, 0, 0, 0',
	X =  2140.450  mm,	Y =   441.871  mm,	Z =  1254.690  mm,
	W =     8.283 deg,	P =   -18.038 deg,	R =   -25.208 deg
   GP2:
	UF : 1, UT : 1,
	J1=   135.000 deg,	J2=     0.000 deg
};
P[141]{
   GP1:
	UF : 1, UT : 1,		CONFIG : 'N U T, 0, 0, 0',
	X =  2140.450  mm,	Y =    13.871  mm,	Z =  1254.689  mm,
	W =     8.283 deg,	P =   -18.038 deg,	R =   -25.208 deg
   GP2:
	UF : 1, UT : 1,
	J1=   135.000 deg,	J2=     0.000 deg
};
P[142]{
   GP1:
	UF : 1, UT : 1,		CONFIG : 'N U T, 0, 0, 0',
	X =  2775.352  mm,	Y =   359.865  mm,	Z =   325.883  mm,
	W =   -20.826 deg,	P =    22.531 deg,	R =    96.055 deg
   GP2:
	UF : 1, UT : 1,
	J1=    90.000 deg,	J2=     0.000 deg
};
P[143]{
   GP1:
	UF : 1, UT : 1,		CONFIG : 'N U T, 0, 0, 0',
	X =  1667.717  mm,	Y =   126.533  mm,	Z =   361.142  mm,
	W =    10.041 deg,	P =    44.100 deg,	R =    14.263 deg
   GP2:
	UF : 1, UT : 1,
	J1=    90.000 deg,	J2=     0.000 deg
};
P[144]{
   GP1:
	UF : 1, UT : 1,		CONFIG : 'N U T, 0, 0, 0',
	X =  2140.450  mm,	Y =    13.871  mm,	Z =  1254.689  mm,
	W =     8.283 deg,	P =   -18.038 deg,	R =   -25.208 deg
   GP2:
	UF : 1, UT : 1,
	J1=   135.000 deg,	J2=     0.000 deg
};
P[145]{
   GP1:
	UF : 1, UT : 1,		CONFIG : 'N U T, 0, 0, 0',
	X =  1669.645  mm,	Y =   204.657  mm,	Z =   362.223  mm,
	W =    10.027 deg,	P =    44.103 deg,	R =    14.252 deg
   GP2:
	UF : 1, UT : 1,
	J1=    90.000 deg,	J2=     0.000 deg
};
P[146]{
   GP1:
	UF : 1, UT : 1,		CONFIG : 'N U T, 0, 0, 0',
	X =  1670.187  mm,	Y =  -130.227  mm,	Z =   362.347  mm,
	W =   -27.010 deg,	P =    37.473 deg,	R =   -36.736 deg
   GP2:
	UF : 1, UT : 1,
	J1=    90.000 deg,	J2=     0.000 deg
};
P[147]{
   GP1:
	UF : 1, UT : 1,		CONFIG : 'N U T, 0, 0, 0',
	X =  2125.819  mm,	Y =    16.776  mm,	Z =  1272.537  mm,
	W =     8.096 deg,	P =   -17.638 deg,	R =   -25.149 deg
   GP2:
	UF : 1, UT : 1,
	J1=   135.000 deg,	J2=     0.000 deg
};
P[148]{
   GP1:
	UF : 1, UT : 1,		CONFIG : 'N U T, 0, 0, 0',
	X =  2115.819  mm,	Y =  -605.300  mm,	Z =  1272.537  mm,
	W =     8.096 deg,	P =   -17.638 deg,	R =   -25.149 deg
   GP2:
	UF : 1, UT : 1,
	J1=   135.000 deg,	J2=     0.000 deg
};
P[149]{
   GP1:
	UF : 1, UT : 1,		CONFIG : 'N U T, 0, 0, 0',
	X =  1671.606  mm,	Y =  -203.809  mm,	Z =   363.549  mm,
	W =   -27.010 deg,	P =    37.473 deg,	R =   -36.736 deg
   GP2:
	UF : 1, UT : 1,
	J1=    90.000 deg,	J2=     0.000 deg
};
P[150]{
   GP1:
	UF : 1, UT : 1,		CONFIG : 'N U T, 0, 0, 0',
	X =  1806.002  mm,	Y =  -392.231  mm,	Z =   828.384  mm,
	W =      .002 deg,	P =      .001 deg,	R =     5.643 deg
   GP2:
	UF : 1, UT : 1,
	J1=    45.000 deg,	J2=     0.000 deg
};
P[151]{
   GP1:
	UF : 1, UT : 1,		CONFIG : 'N U T, 0, 0, 0',
	X =  2140.208  mm,	Y =  -654.090  mm,	Z =  1313.833  mm,
	W =    10.028 deg,	P =   -21.460 deg,	R =   -25.796 deg
   GP2:
	UF : 1, UT : 1,
	J1=   135.000 deg,	J2=     0.000 deg
};
P[152]{
   GP1:
	UF : 1, UT : 1,		CONFIG : 'N U T, 0, 0, 0',
	X =  1423.602  mm,	Y =  -633.435  mm,	Z =  1512.519  mm,
	W =    10.028 deg,	P =   -21.460 deg,	R =   -25.796 deg
   GP2:
	UF : 1, UT : 1,
	J1=   135.000 deg,	J2=     0.000 deg
};
P[153]{
   GP1:
	UF : 1, UT : 1,		CONFIG : 'N U B, 0, 0, 0',
	X =   357.030  mm,	Y =     -.134  mm,	Z =  2422.493  mm,
	W =     -.020 deg,	P =   -39.773 deg,	R =      .020 deg
   GP2:
	UF : 1, UT : 1,
	J1=     0.000 deg,	J2=   180.000 deg
};
P[154]{
   GP1:
	UF : 1, UT : 1,		CONFIG : 'N U T, 0, 0, 0',
	X =  2120.617  mm,	Y =   114.231  mm,	Z =   454.022  mm,
	W =     -.010 deg,	P =    45.000 deg,	R =   -90.000 deg
   GP2:
	UF : 1, UT : 1,
	J1=     0.000 deg,	J2=   180.000 deg
};
P[155]{
   GP1:
	UF : 1, UT : 1,		CONFIG : 'N U T, 0, 0, 0',
	X =  2322.538  mm,	Y =   282.923  mm,	Z =   407.108  mm,
	W =    44.356 deg,	P =     8.527 deg,	R =    -8.608 deg
   GP2:
	UF : 1, UT : 1,
	J1=     0.000 deg,	J2=   180.000 deg
};
P[156]{
   GP1:
	UF : 1, UT : 1,		CONFIG : 'N U T, 0, 0, 0',
	X =  1807.388  mm,	Y =  -132.355  mm,	Z =   830.745  mm,
	W =      .017 deg,	P =      .003 deg,	R =     5.640 deg
   GP2:
	UF : 1, UT : 1,
	J1=    45.000 deg,	J2=     0.000 deg
};
P[157]{
   GP1:
	UF : 1, UT : 1,		CONFIG : 'N U T, 0, 0, 0',
	X =  1805.255  mm,	Y =   387.768  mm,	Z =   830.985  mm,
	W =     -.593 deg,	P =    -5.980 deg,	R =     5.674 deg
   GP2:
	UF : 1, UT : 1,
	J1=    45.000 deg,	J2=     0.000 deg
};
P[158]{
   GP1:
	UF : 1, UT : 1,		CONFIG : 'N U T, 0, 0, 0',
	X =  1807.100  mm,	Y =   128.882  mm,	Z =   831.212  mm,
	W =     -.593 deg,	P =    -5.980 deg,	R =     5.674 deg
   GP2:
	UF : 1, UT : 1,
	J1=    45.000 deg,	J2=     0.000 deg
};
P[159]{
   GP1:
	UF : 1, UT : 1,		CONFIG : 'N U T, 0, 0, 0',
	X =  2337.926  mm,	Y =   299.816  mm,	Z =   380.534  mm,
	W =    43.107 deg,	P =    14.444 deg,	R =    14.426 deg
   GP2:
	UF : 1, UT : 1,
	J1=     0.000 deg,	J2=   180.000 deg
};
P[160]{
   GP1:
	UF : 1, UT : 1,		CONFIG : 'N U T, 0, 0, 0',
	X =  2369.612  mm,	Y =  -152.146  mm,	Z =   450.842  mm,
	W =   -35.390 deg,	P =     -.015 deg,	R =    11.717 deg
   GP2:
	UF : 1, UT : 1,
	J1=     0.000 deg,	J2=   180.000 deg
};
P[161]{
   GP1:
	UF : 1, UT : 1,		CONFIG : 'N U T, 0, 0, 0',
	X =  2324.098  mm,	Y =  -366.142  mm,	Z =   356.893  mm,
	W =   -26.270 deg,	P =   -24.616 deg,	R =   -28.424 deg
   GP2:
	UF : 1, UT : 1,
	J1=     0.000 deg,	J2=   180.000 deg
};
P[162]{
   GP1:
	UF : 1, UT : 1,		CONFIG : 'N U T, 0, 0, 0',
	X =  2125.842  mm,	Y =   644.021  mm,	Z =  1177.221  mm,
	W =     1.340 deg,	P =     1.267 deg,	R =   -23.862 deg
   GP2:
	UF : 1, UT : 1,
	J1=   135.000 deg,	J2=     0.000 deg
};
P[163]{
   GP1:
	UF : 1, UT : 1,		CONFIG : 'N U T, 0, 0, 0',
	X =  2126.827  mm,	Y =   449.706  mm,	Z =  1179.015  mm,
	W =      .101 deg,	P =     -.251 deg,	R =   -23.878 deg
   GP2:
	UF : 1, UT : 1,
	J1=   135.000 deg,	J2=     0.000 deg
};
P[164]{
   GP1:
	UF : 1, UT : 1,		CONFIG : 'N U T, 0, 0, 0',
	X =  2126.970  mm,	Y =   444.920  mm,	Z =  1178.159  mm,
	W =    -7.000 deg,	P =    -3.382 deg,	R =   -23.652 deg
   GP2:
	UF : 1, UT : 1,
	J1=   135.000 deg,	J2=     0.000 deg
};
P[165]{
   GP1:
	UF : 1, UT : 1,		CONFIG : 'N U T, 0, 0, 0',
	X =  2347.623  mm,	Y =  -252.998  mm,	Z =   505.500  mm,
	W =   -41.361 deg,	P =   -19.588 deg,	R =    -2.703 deg
   GP2:
	UF : 1, UT : 1,
	J1=     0.000 deg,	J2=   180.000 deg
};
P[166]{
   GP1:
	UF : 1, UT : 1,		CONFIG : 'N U T, 0, 0, 0',
	X =  2072.623  mm,	Y =  -178.998  mm,	Z =   505.500  mm,
	W =    32.971 deg,	P =    25.781 deg,	R =  -125.417 deg
   GP2:
	UF : 1, UT : 1,
	J1=     0.000 deg,	J2=   180.000 deg
};
P[167]{
   GP1:
	UF : 1, UT : 1,		CONFIG : 'N U T, 0, 0, 0',
	X =  2278.079  mm,	Y =  -225.854  mm,	Z =   -19.500  mm,
	W =    32.971 deg,	P =    25.781 deg,	R =  -125.417 deg
   GP2:
	UF : 1, UT : 1,
	J1=     0.000 deg,	J2=   180.000 deg
};
P[168]{
   GP1:
	UF : 1, UT : 1,		CONFIG : 'N U T, 0, 0, 0',
	X =  2111.886  mm,	Y =     7.673  mm,	Z =  1193.435  mm,
	W =    -1.732 deg,	P =    -2.297 deg,	R =   -23.799 deg
   GP2:
	UF : 1, UT : 1,
	J1=   135.000 deg,	J2=     0.000 deg
};
P[169]{
   GP1:
	UF : 1, UT : 1,		CONFIG : 'N U T, 0, 0, 0',
	X =  2111.696  mm,	Y =  -402.392  mm,	Z =  1193.417  mm,
	W =    -1.735 deg,	P =    -2.297 deg,	R =   -23.794 deg
   GP2:
	UF : 1, UT : 1,
	J1=   135.000 deg,	J2=     0.000 deg
};
P[170]{
   GP1:
	UF : 1, UT : 1,		CONFIG : 'N U T, 0, 0, 0',
	X =  1460.901  mm,	Y =  -124.727  mm,	Z =   173.177  mm,
	W =   -18.859 deg,	P =    44.384 deg,	R =   163.367 deg
   GP2:
	UF : 1, UT : 1,
	J1=     0.000 deg,	J2=   180.000 deg
};
P[171]{
   GP1:
	UF : 1, UT : 1,		CONFIG : 'N U T, 0, 0, 0',
	X =  1549.299  mm,	Y =  -552.174  mm,	Z =   106.967  mm,
	W =   -29.293 deg,	P =    36.031 deg,	R =   140.482 deg
   GP2:
	UF : 1, UT : 1,
